	bArm2VertStn4Down_00 AT %MX26516.0 : BOOL;
	bArm2VertStn4Down_01 AT %MX26516.1 : BOOL;
	bArm2VertStn4Down_02 AT %MX26516.2 : BOOL;
	bArm2VertStn4Down_03 AT %MX26516.3 : BOOL;
	bArm2VertStn4Down_04 AT %MX26516.4 : BOOL;
	bArm2VertStn4Down_05 AT %MX26516.5 : BOOL;
	bArm2VertStn4Down_06 AT %MX26516.6 : BOOL;
	bArm2VertStn4Down_07 AT %MX26516.7 : BOOL;
	bArm2VertStn4Down_08 AT %MX26516.8 : BOOL;
	bArm2VertStn4Down_09 AT %MX26516.9 : BOOL;
	bArm2VertStn4Down_10 AT %MX26516.10 : BOOL;
	bArm2VertStn4Down_11 AT %MX26516.11 : BOOL;
	bArm2VertStn4Down_12 AT %MX26516.12 : BOOL;
	bArm2VertStn4Down_13 AT %MX26516.13 : BOOL;
	bArm2VertStn4Down_14 AT %MX26516.14 : BOOL;
	bArm2VertStn4Down_15 AT %MX26516.15 : BOOL;
	bArm2VertStn4Down_16 AT %MX26516.16 : BOOL;
	bArm2VertStn4Down_17 AT %MX26516.17 : BOOL;
	bArm2VertStn4Down_18 AT %MX26516.18 : BOOL;
	bArm2VertStn4Down_19 AT %MX26516.19 : BOOL;
	bArm2VertStn4Down_20 AT %MX26516.20 : BOOL;
	bArm2VertStn4Down_21 AT %MX26516.21 : BOOL;
	bArm2VertStn4Down_22 AT %MX26516.22 : BOOL;
	bArm2VertStn4Down_23 AT %MX26516.23 : BOOL;
	bArm2VertStn4Down_24 AT %MX26516.24 : BOOL;
	bArm2VertStn4Down_25 AT %MX26516.25 : BOOL;
	bArm2VertStn4Down_26 AT %MX26516.26 : BOOL;
	bArm2VertStn4Down_27 AT %MX26516.27 : BOOL;
	bArm2VertStn4Down_28 AT %MX26516.28 : BOOL;
	bArm2VertStn4Down_29 AT %MX26516.29 : BOOL;
	bArm2VertStn4Down_30 AT %MX26516.30 : BOOL;
	bArm2VertStn4Down_31 AT %MX26516.31 : BOOL;

	bArm2VertStn5Down_00 AT %MX26520.0 : BOOL;
	bArm2VertStn5Down_01 AT %MX26520.1 : BOOL;
	bArm2VertStn5Down_02 AT %MX26520.2 : BOOL;
	bArm2VertStn5Down_03 AT %MX26520.3 : BOOL;
	bArm2VertStn5Down_04 AT %MX26520.4 : BOOL;
	bArm2VertStn5Down_05 AT %MX26520.5 : BOOL;
	bArm2VertStn5Down_06 AT %MX26520.6 : BOOL;
	bArm2VertStn5Down_07 AT %MX26520.7 : BOOL;
	bArm2VertStn5Down_08 AT %MX26520.8 : BOOL;
	bArm2VertStn5Down_09 AT %MX26520.9 : BOOL;
	bArm2VertStn5Down_10 AT %MX26520.10 : BOOL;
	bArm2VertStn5Down_11 AT %MX26520.11 : BOOL;
	bArm2VertStn5Down_12 AT %MX26520.12 : BOOL;
	bArm2VertStn5Down_13 AT %MX26520.13 : BOOL;
	bArm2VertStn5Down_14 AT %MX26520.14 : BOOL;
	bArm2VertStn5Down_15 AT %MX26520.15 : BOOL;
	bArm2VertStn5Down_16 AT %MX26520.16 : BOOL;
	bArm2VertStn5Down_17 AT %MX26520.17 : BOOL;
	bArm2VertStn5Down_18 AT %MX26520.18 : BOOL;
	bArm2VertStn5Down_19 AT %MX26520.19 : BOOL;
	bArm2VertStn5Down_20 AT %MX26520.20 : BOOL;
	bArm2VertStn5Down_21 AT %MX26520.21 : BOOL;
	bArm2VertStn5Down_22 AT %MX26520.22 : BOOL;
	bArm2VertStn5Down_23 AT %MX26520.23 : BOOL;
	bArm2VertStn5Down_24 AT %MX26520.24 : BOOL;
	bArm2VertStn5Down_25 AT %MX26520.25 : BOOL;
	bArm2VertStn5Down_26 AT %MX26520.26 : BOOL;
	bArm2VertStn5Down_27 AT %MX26520.27 : BOOL;
	bArm2VertStn5Down_28 AT %MX26520.28 : BOOL;
	bArm2VertStn5Down_29 AT %MX26520.29 : BOOL;
	bArm2VertStn5Down_30 AT %MX26520.30 : BOOL;
	bArm2VertStn5Down_31 AT %MX26520.31 : BOOL;

	bArm2VertStn6Down_00 AT %MX26524.0 : BOOL;
	bArm2VertStn6Down_01 AT %MX26524.1 : BOOL;
	bArm2VertStn6Down_02 AT %MX26524.2 : BOOL;
	bArm2VertStn6Down_03 AT %MX26524.3 : BOOL;
	bArm2VertStn6Down_04 AT %MX26524.4 : BOOL;
	bArm2VertStn6Down_05 AT %MX26524.5 : BOOL;
	bArm2VertStn6Down_06 AT %MX26524.6 : BOOL;
	bArm2VertStn6Down_07 AT %MX26524.7 : BOOL;
	bArm2VertStn6Down_08 AT %MX26524.8 : BOOL;
	bArm2VertStn6Down_09 AT %MX26524.9 : BOOL;
	bArm2VertStn6Down_10 AT %MX26524.10 : BOOL;
	bArm2VertStn6Down_11 AT %MX26524.11 : BOOL;
	bArm2VertStn6Down_12 AT %MX26524.12 : BOOL;
	bArm2VertStn6Down_13 AT %MX26524.13 : BOOL;
	bArm2VertStn6Down_14 AT %MX26524.14 : BOOL;
	bArm2VertStn6Down_15 AT %MX26524.15 : BOOL;
	bArm2VertStn6Down_16 AT %MX26524.16 : BOOL;
	bArm2VertStn6Down_17 AT %MX26524.17 : BOOL;
	bArm2VertStn6Down_18 AT %MX26524.18 : BOOL;
	bArm2VertStn6Down_19 AT %MX26524.19 : BOOL;
	bArm2VertStn6Down_20 AT %MX26524.20 : BOOL;
	bArm2VertStn6Down_21 AT %MX26524.21 : BOOL;
	bArm2VertStn6Down_22 AT %MX26524.22 : BOOL;
	bArm2VertStn6Down_23 AT %MX26524.23 : BOOL;
	bArm2VertStn6Down_24 AT %MX26524.24 : BOOL;
	bArm2VertStn6Down_25 AT %MX26524.25 : BOOL;
	bArm2VertStn6Down_26 AT %MX26524.26 : BOOL;
	bArm2VertStn6Down_27 AT %MX26524.27 : BOOL;
	bArm2VertStn6Down_28 AT %MX26524.28 : BOOL;
	bArm2VertStn6Down_29 AT %MX26524.29 : BOOL;
	bArm2VertStn6Down_30 AT %MX26524.30 : BOOL;
	bArm2VertStn6Down_31 AT %MX26524.31 : BOOL;

	bArm2VertStn7Down_00 AT %MX26528.0 : BOOL;
	bArm2VertStn7Down_01 AT %MX26528.1 : BOOL;
	bArm2VertStn7Down_02 AT %MX26528.2 : BOOL;
	bArm2VertStn7Down_03 AT %MX26528.3 : BOOL;
	bArm2VertStn7Down_04 AT %MX26528.4 : BOOL;
	bArm2VertStn7Down_05 AT %MX26528.5 : BOOL;
	bArm2VertStn7Down_06 AT %MX26528.6 : BOOL;
	bArm2VertStn7Down_07 AT %MX26528.7 : BOOL;
	bArm2VertStn7Down_08 AT %MX26528.8 : BOOL;
	bArm2VertStn7Down_09 AT %MX26528.9 : BOOL;
	bArm2VertStn7Down_10 AT %MX26528.10 : BOOL;
	bArm2VertStn7Down_11 AT %MX26528.11 : BOOL;
	bArm2VertStn7Down_12 AT %MX26528.12 : BOOL;
	bArm2VertStn7Down_13 AT %MX26528.13 : BOOL;
	bArm2VertStn7Down_14 AT %MX26528.14 : BOOL;
	bArm2VertStn7Down_15 AT %MX26528.15 : BOOL;
	bArm2VertStn7Down_16 AT %MX26528.16 : BOOL;
	bArm2VertStn7Down_17 AT %MX26528.17 : BOOL;
	bArm2VertStn7Down_18 AT %MX26528.18 : BOOL;
	bArm2VertStn7Down_19 AT %MX26528.19 : BOOL;
	bArm2VertStn7Down_20 AT %MX26528.20 : BOOL;
	bArm2VertStn7Down_21 AT %MX26528.21 : BOOL;
	bArm2VertStn7Down_22 AT %MX26528.22 : BOOL;
	bArm2VertStn7Down_23 AT %MX26528.23 : BOOL;
	bArm2VertStn7Down_24 AT %MX26528.24 : BOOL;
	bArm2VertStn7Down_25 AT %MX26528.25 : BOOL;
	bArm2VertStn7Down_26 AT %MX26528.26 : BOOL;
	bArm2VertStn7Down_27 AT %MX26528.27 : BOOL;
	bArm2VertStn7Down_28 AT %MX26528.28 : BOOL;
	bArm2VertStn7Down_29 AT %MX26528.29 : BOOL;
	bArm2VertStn7Down_30 AT %MX26528.30 : BOOL;
	bArm2VertStn7Down_31 AT %MX26528.31 : BOOL;

	bArm2VertStn8Down_00 AT %MX26532.0 : BOOL;
	bArm2VertStn8Down_01 AT %MX26532.1 : BOOL;
	bArm2VertStn8Down_02 AT %MX26532.2 : BOOL;
	bArm2VertStn8Down_03 AT %MX26532.3 : BOOL;
	bArm2VertStn8Down_04 AT %MX26532.4 : BOOL;
	bArm2VertStn8Down_05 AT %MX26532.5 : BOOL;
	bArm2VertStn8Down_06 AT %MX26532.6 : BOOL;
	bArm2VertStn8Down_07 AT %MX26532.7 : BOOL;
	bArm2VertStn8Down_08 AT %MX26532.8 : BOOL;
	bArm2VertStn8Down_09 AT %MX26532.9 : BOOL;
	bArm2VertStn8Down_10 AT %MX26532.10 : BOOL;
	bArm2VertStn8Down_11 AT %MX26532.11 : BOOL;
	bArm2VertStn8Down_12 AT %MX26532.12 : BOOL;
	bArm2VertStn8Down_13 AT %MX26532.13 : BOOL;
	bArm2VertStn8Down_14 AT %MX26532.14 : BOOL;
	bArm2VertStn8Down_15 AT %MX26532.15 : BOOL;
	bArm2VertStn8Down_16 AT %MX26532.16 : BOOL;
	bArm2VertStn8Down_17 AT %MX26532.17 : BOOL;
	bArm2VertStn8Down_18 AT %MX26532.18 : BOOL;
	bArm2VertStn8Down_19 AT %MX26532.19 : BOOL;
	bArm2VertStn8Down_20 AT %MX26532.20 : BOOL;
	bArm2VertStn8Down_21 AT %MX26532.21 : BOOL;
	bArm2VertStn8Down_22 AT %MX26532.22 : BOOL;
	bArm2VertStn8Down_23 AT %MX26532.23 : BOOL;
	bArm2VertStn8Down_24 AT %MX26532.24 : BOOL;
	bArm2VertStn8Down_25 AT %MX26532.25 : BOOL;
	bArm2VertStn8Down_26 AT %MX26532.26 : BOOL;
	bArm2VertStn8Down_27 AT %MX26532.27 : BOOL;
	bArm2VertStn8Down_28 AT %MX26532.28 : BOOL;
	bArm2VertStn8Down_29 AT %MX26532.29 : BOOL;
	bArm2VertStn8Down_30 AT %MX26532.30 : BOOL;
	bArm2VertStn8Down_31 AT %MX26532.31 : BOOL;

	bArm2VertStn9Down_00 AT %MX26536.0 : BOOL;
	bArm2VertStn9Down_01 AT %MX26536.1 : BOOL;
	bArm2VertStn9Down_02 AT %MX26536.2 : BOOL;
	bArm2VertStn9Down_03 AT %MX26536.3 : BOOL;
	bArm2VertStn9Down_04 AT %MX26536.4 : BOOL;
	bArm2VertStn9Down_05 AT %MX26536.5 : BOOL;
	bArm2VertStn9Down_06 AT %MX26536.6 : BOOL;
	bArm2VertStn9Down_07 AT %MX26536.7 : BOOL;
	bArm2VertStn9Down_08 AT %MX26536.8 : BOOL;
	bArm2VertStn9Down_09 AT %MX26536.9 : BOOL;
	bArm2VertStn9Down_10 AT %MX26536.10 : BOOL;
	bArm2VertStn9Down_11 AT %MX26536.11 : BOOL;
	bArm2VertStn9Down_12 AT %MX26536.12 : BOOL;
	bArm2VertStn9Down_13 AT %MX26536.13 : BOOL;
	bArm2VertStn9Down_14 AT %MX26536.14 : BOOL;
	bArm2VertStn9Down_15 AT %MX26536.15 : BOOL;
	bArm2VertStn9Down_16 AT %MX26536.16 : BOOL;
	bArm2VertStn9Down_17 AT %MX26536.17 : BOOL;
	bArm2VertStn9Down_18 AT %MX26536.18 : BOOL;
	bArm2VertStn9Down_19 AT %MX26536.19 : BOOL;
	bArm2VertStn9Down_20 AT %MX26536.20 : BOOL;
	bArm2VertStn9Down_21 AT %MX26536.21 : BOOL;
	bArm2VertStn9Down_22 AT %MX26536.22 : BOOL;
	bArm2VertStn9Down_23 AT %MX26536.23 : BOOL;
	bArm2VertStn9Down_24 AT %MX26536.24 : BOOL;
	bArm2VertStn9Down_25 AT %MX26536.25 : BOOL;
	bArm2VertStn9Down_26 AT %MX26536.26 : BOOL;
	bArm2VertStn9Down_27 AT %MX26536.27 : BOOL;
	bArm2VertStn9Down_28 AT %MX26536.28 : BOOL;
	bArm2VertStn9Down_29 AT %MX26536.29 : BOOL;
	bArm2VertStn9Down_30 AT %MX26536.30 : BOOL;
	bArm2VertStn9Down_31 AT %MX26536.31 : BOOL;

	bArm2VertStn10Down_00 AT %MX26540.0 : BOOL;
	bArm2VertStn10Down_01 AT %MX26540.1 : BOOL;
	bArm2VertStn10Down_02 AT %MX26540.2 : BOOL;
	bArm2VertStn10Down_03 AT %MX26540.3 : BOOL;
	bArm2VertStn10Down_04 AT %MX26540.4 : BOOL;
	bArm2VertStn10Down_05 AT %MX26540.5 : BOOL;
	bArm2VertStn10Down_06 AT %MX26540.6 : BOOL;
	bArm2VertStn10Down_07 AT %MX26540.7 : BOOL;
	bArm2VertStn10Down_08 AT %MX26540.8 : BOOL;
	bArm2VertStn10Down_09 AT %MX26540.9 : BOOL;
	bArm2VertStn10Down_10 AT %MX26540.10 : BOOL;
	bArm2VertStn10Down_11 AT %MX26540.11 : BOOL;
	bArm2VertStn10Down_12 AT %MX26540.12 : BOOL;
	bArm2VertStn10Down_13 AT %MX26540.13 : BOOL;
	bArm2VertStn10Down_14 AT %MX26540.14 : BOOL;
	bArm2VertStn10Down_15 AT %MX26540.15 : BOOL;
	bArm2VertStn10Down_16 AT %MX26540.16 : BOOL;
	bArm2VertStn10Down_17 AT %MX26540.17 : BOOL;
	bArm2VertStn10Down_18 AT %MX26540.18 : BOOL;
	bArm2VertStn10Down_19 AT %MX26540.19 : BOOL;
	bArm2VertStn10Down_20 AT %MX26540.20 : BOOL;
	bArm2VertStn10Down_21 AT %MX26540.21 : BOOL;
	bArm2VertStn10Down_22 AT %MX26540.22 : BOOL;
	bArm2VertStn10Down_23 AT %MX26540.23 : BOOL;
	bArm2VertStn10Down_24 AT %MX26540.24 : BOOL;
	bArm2VertStn10Down_25 AT %MX26540.25 : BOOL;
	bArm2VertStn10Down_26 AT %MX26540.26 : BOOL;
	bArm2VertStn10Down_27 AT %MX26540.27 : BOOL;
	bArm2VertStn10Down_28 AT %MX26540.28 : BOOL;
	bArm2VertStn10Down_29 AT %MX26540.29 : BOOL;
	bArm2VertStn10Down_30 AT %MX26540.30 : BOOL;
	bArm2VertStn10Down_31 AT %MX26540.31 : BOOL;

	bArm2VertStn11Down_00 AT %MX26544.0 : BOOL;
	bArm2VertStn11Down_01 AT %MX26544.1 : BOOL;
	bArm2VertStn11Down_02 AT %MX26544.2 : BOOL;
	bArm2VertStn11Down_03 AT %MX26544.3 : BOOL;
	bArm2VertStn11Down_04 AT %MX26544.4 : BOOL;
	bArm2VertStn11Down_05 AT %MX26544.5 : BOOL;
	bArm2VertStn11Down_06 AT %MX26544.6 : BOOL;
	bArm2VertStn11Down_07 AT %MX26544.7 : BOOL;
	bArm2VertStn11Down_08 AT %MX26544.8 : BOOL;
	bArm2VertStn11Down_09 AT %MX26544.9 : BOOL;
	bArm2VertStn11Down_10 AT %MX26544.10 : BOOL;
	bArm2VertStn11Down_11 AT %MX26544.11 : BOOL;
	bArm2VertStn11Down_12 AT %MX26544.12 : BOOL;
	bArm2VertStn11Down_13 AT %MX26544.13 : BOOL;
	bArm2VertStn11Down_14 AT %MX26544.14 : BOOL;
	bArm2VertStn11Down_15 AT %MX26544.15 : BOOL;
	bArm2VertStn11Down_16 AT %MX26544.16 : BOOL;
	bArm2VertStn11Down_17 AT %MX26544.17 : BOOL;
	bArm2VertStn11Down_18 AT %MX26544.18 : BOOL;
	bArm2VertStn11Down_19 AT %MX26544.19 : BOOL;
	bArm2VertStn11Down_20 AT %MX26544.20 : BOOL;
	bArm2VertStn11Down_21 AT %MX26544.21 : BOOL;
	bArm2VertStn11Down_22 AT %MX26544.22 : BOOL;
	bArm2VertStn11Down_23 AT %MX26544.23 : BOOL;
	bArm2VertStn11Down_24 AT %MX26544.24 : BOOL;
	bArm2VertStn11Down_25 AT %MX26544.25 : BOOL;
	bArm2VertStn11Down_26 AT %MX26544.26 : BOOL;
	bArm2VertStn11Down_27 AT %MX26544.27 : BOOL;
	bArm2VertStn11Down_28 AT %MX26544.28 : BOOL;
	bArm2VertStn11Down_29 AT %MX26544.29 : BOOL;
	bArm2VertStn11Down_30 AT %MX26544.30 : BOOL;
	bArm2VertStn11Down_31 AT %MX26544.31 : BOOL;

	bArm2VertStn12Down_00 AT %MX26548.0 : BOOL;
	bArm2VertStn12Down_01 AT %MX26548.1 : BOOL;
	bArm2VertStn12Down_02 AT %MX26548.2 : BOOL;
	bArm2VertStn12Down_03 AT %MX26548.3 : BOOL;
	bArm2VertStn12Down_04 AT %MX26548.4 : BOOL;
	bArm2VertStn12Down_05 AT %MX26548.5 : BOOL;
	bArm2VertStn12Down_06 AT %MX26548.6 : BOOL;
	bArm2VertStn12Down_07 AT %MX26548.7 : BOOL;
	bArm2VertStn12Down_08 AT %MX26548.8 : BOOL;
	bArm2VertStn12Down_09 AT %MX26548.9 : BOOL;
	bArm2VertStn12Down_10 AT %MX26548.10 : BOOL;
	bArm2VertStn12Down_11 AT %MX26548.11 : BOOL;
	bArm2VertStn12Down_12 AT %MX26548.12 : BOOL;
	bArm2VertStn12Down_13 AT %MX26548.13 : BOOL;
	bArm2VertStn12Down_14 AT %MX26548.14 : BOOL;
	bArm2VertStn12Down_15 AT %MX26548.15 : BOOL;
	bArm2VertStn12Down_16 AT %MX26548.16 : BOOL;
	bArm2VertStn12Down_17 AT %MX26548.17 : BOOL;
	bArm2VertStn12Down_18 AT %MX26548.18 : BOOL;
	bArm2VertStn12Down_19 AT %MX26548.19 : BOOL;
	bArm2VertStn12Down_20 AT %MX26548.20 : BOOL;
	bArm2VertStn12Down_21 AT %MX26548.21 : BOOL;
	bArm2VertStn12Down_22 AT %MX26548.22 : BOOL;
	bArm2VertStn12Down_23 AT %MX26548.23 : BOOL;
	bArm2VertStn12Down_24 AT %MX26548.24 : BOOL;
	bArm2VertStn12Down_25 AT %MX26548.25 : BOOL;
	bArm2VertStn12Down_26 AT %MX26548.26 : BOOL;
	bArm2VertStn12Down_27 AT %MX26548.27 : BOOL;
	bArm2VertStn12Down_28 AT %MX26548.28 : BOOL;
	bArm2VertStn12Down_29 AT %MX26548.29 : BOOL;
	bArm2VertStn12Down_30 AT %MX26548.30 : BOOL;
	bArm2VertStn12Down_31 AT %MX26548.31 : BOOL;


(* xxxxxxxxxxxxxxxxxxxxxxxxxxxxxxxxxxxxxxx Lifter xxxxxxxxxxxxxxxxxxxxxxxxxxxxxxxxxxxxxxx*)
(*========= Up/Down LifterUp BOOL LINK with %MX31000-  =========*)

	bSlowPull2LifterStn1Up_00 AT %MX31004.0 : BOOL;
	bSlowPull2LifterStn1Up_01 AT %MX31004.1 : BOOL;
	bSlowPull2LifterStn1Up_02 AT %MX31004.2 : BOOL;
	bSlowPull2LifterStn1Up_03 AT %MX31004.3 : BOOL;
	bSlowPull2LifterStn1Up_04 AT %MX31004.4 : BOOL;
	bSlowPull2LifterStn1Up_05 AT %MX31004.5 : BOOL;
	bSlowPull2LifterStn1Up_06 AT %MX31004.6 : BOOL;
	bSlowPull2LifterStn1Up_07 AT %MX31004.7 : BOOL;
	bSlowPull2LifterStn1Up_08 AT %MX31004.8 : BOOL;
	bSlowPull2LifterStn1Up_09 AT %MX31004.9 : BOOL;
	bSlowPull2LifterStn1Up_10 AT %MX31004.10 : BOOL;
	bSlowPull2LifterStn1Up_11 AT %MX31004.11 : BOOL;
	bSlowPull2LifterStn1Up_12 AT %MX31004.12 : BOOL;
	bSlowPull2LifterStn1Up_13 AT %MX31004.13 : BOOL;
	bSlowPull2LifterStn1Up_14 AT %MX31004.14 : BOOL;
	bSlowPull2LifterStn1Up_15 AT %MX31004.15 : BOOL;
	bSlowPull2LifterStn1Up_16 AT %MX31004.16 : BOOL;
	bSlowPull2LifterStn1Up_17 AT %MX31004.17 : BOOL;
	bSlowPull2LifterStn1Up_18 AT %MX31004.18 : BOOL;
	bSlowPull2LifterStn1Up_19 AT %MX31004.19 : BOOL;
	bSlowPull2LifterStn1Up_20 AT %MX31004.20 : BOOL;
	bSlowPull2LifterStn1Up_21 AT %MX31004.21 : BOOL;
	bSlowPull2LifterStn1Up_22 AT %MX31004.22 : BOOL;
	bSlowPull2LifterStn1Up_23 AT %MX31004.23 : BOOL;
	bSlowPull2LifterStn1Up_24 AT %MX31004.24 : BOOL;
	bSlowPull2LifterStn1Up_25 AT %MX31004.25 : BOOL;
	bSlowPull2LifterStn1Up_26 AT %MX31004.26 : BOOL;
	bSlowPull2LifterStn1Up_27 AT %MX31004.27 : BOOL;
	bSlowPull2LifterStn1Up_28 AT %MX31004.28 : BOOL;
	bSlowPull2LifterStn1Up_29 AT %MX31004.29 : BOOL;
	bSlowPull2LifterStn1Up_30 AT %MX31004.30 : BOOL;
	bSlowPull2LifterStn1Up_31 AT %MX31004.31 : BOOL;

	bSlowPull2LifterStn2Up_00 AT %MX31008.0 : BOOL;
	bSlowPull2LifterStn2Up_01 AT %MX31008.1 : BOOL;
	bSlowPull2LifterStn2Up_02 AT %MX31008.2 : BOOL;
	bSlowPull2LifterStn2Up_03 AT %MX31008.3 : BOOL;
	bSlowPull2LifterStn2Up_04 AT %MX31008.4 : BOOL;
	bSlowPull2LifterStn2Up_05 AT %MX31008.5 : BOOL;
	bSlowPull2LifterStn2Up_06 AT %MX31008.6 : BOOL;
	bSlowPull2LifterStn2Up_07 AT %MX31008.7 : BOOL;
	bSlowPull2LifterStn2Up_08 AT %MX31008.8 : BOOL;
	bSlowPull2LifterStn2Up_09 AT %MX31008.9 : BOOL;
	bSlowPull2LifterStn2Up_10 AT %MX31008.10 : BOOL;
	bSlowPull2LifterStn2Up_11 AT %MX31008.11 : BOOL;
	bSlowPull2LifterStn2Up_12 AT %MX31008.12 : BOOL;
	bSlowPull2LifterStn2Up_13 AT %MX31008.13 : BOOL;
	bSlowPull2LifterStn2Up_14 AT %MX31008.14 : BOOL;
	bSlowPull2LifterStn2Up_15 AT %MX31008.15 : BOOL;
	bSlowPull2LifterStn2Up_16 AT %MX31008.16 : BOOL;
	bSlowPull2LifterStn2Up_17 AT %MX31008.17 : BOOL;
	bSlowPull2LifterStn2Up_18 AT %MX31008.18 : BOOL;
	bSlowPull2LifterStn2Up_19 AT %MX31008.19 : BOOL;
	bSlowPull2LifterStn2Up_20 AT %MX31008.20 : BOOL;
	bSlowPull2LifterStn2Up_21 AT %MX31008.21 : BOOL;
	bSlowPull2LifterStn2Up_22 AT %MX31008.22 : BOOL;
	bSlowPull2LifterStn2Up_23 AT %MX31008.23 : BOOL;
	bSlowPull2LifterStn2Up_24 AT %MX31008.24 : BOOL;
	bSlowPull2LifterStn2Up_25 AT %MX31008.25 : BOOL;
	bSlowPull2LifterStn2Up_26 AT %MX31008.26 : BOOL;
	bSlowPull2LifterStn2Up_27 AT %MX31008.27 : BOOL;
	bSlowPull2LifterStn2Up_28 AT %MX31008.28 : BOOL;
	bSlowPull2LifterStn2Up_29 AT %MX31008.29 : BOOL;
	bSlowPull2LifterStn2Up_30 AT %MX31008.30 : BOOL;
	bSlowPull2LifterStn2Up_31 AT %MX31008.31 : BOOL;

	bSlowPull2LifterStn3Up_00 AT %MX31012.0 : BOOL;
	bSlowPull2LifterStn3Up_01 AT %MX31012.1 : BOOL;
	bSlowPull2LifterStn3Up_02 AT %MX31012.2 : BOOL;
	bSlowPull2LifterStn3Up_03 AT %MX31012.3 : BOOL;
	bSlowPull2LifterStn3Up_04 AT %MX31012.4 : BOOL;
	bSlowPull2LifterStn3Up_05 AT %MX31012.5 : BOOL;
	bSlowPull2LifterStn3Up_06 AT %MX31012.6 : BOOL;
	bSlowPull2LifterStn3Up_07 AT %MX31012.7 : BOOL;
	bSlowPull2LifterStn3Up_08 AT %MX31012.8 : BOOL;
	bSlowPull2LifterStn3Up_09 AT %MX31012.9 : BOOL;
	bSlowPull2LifterStn3Up_10 AT %MX31012.10 : BOOL;
	bSlowPull2LifterStn3Up_11 AT %MX31012.11 : BOOL;
	bSlowPull2LifterStn3Up_12 AT %MX31012.12 : BOOL;
	bSlowPull2LifterStn3Up_13 AT %MX31012.13 : BOOL;
	bSlowPull2LifterStn3Up_14 AT %MX31012.14 : BOOL;
	bSlowPull2LifterStn3Up_15 AT %MX31012.15 : BOOL;
	bSlowPull2LifterStn3Up_16 AT %MX31012.16 : BOOL;
	bSlowPull2LifterStn3Up_17 AT %MX31012.17 : BOOL;
	bSlowPull2LifterStn3Up_18 AT %MX31012.18 : BOOL;
	bSlowPull2LifterStn3Up_19 AT %MX31012.19 : BOOL;
	bSlowPull2LifterStn3Up_20 AT %MX31012.20 : BOOL;
	bSlowPull2LifterStn3Up_21 AT %MX31012.21 : BOOL;
	bSlowPull2LifterStn3Up_22 AT %MX31012.22 : BOOL;
	bSlowPull2LifterStn3Up_23 AT %MX31012.23 : BOOL;
	bSlowPull2LifterStn3Up_24 AT %MX31012.24 : BOOL;
	bSlowPull2LifterStn3Up_25 AT %MX31012.25 : BOOL;
	bSlowPull2LifterStn3Up_26 AT %MX31012.26 : BOOL;
	bSlowPull2LifterStn3Up_27 AT %MX31012.27 : BOOL;
	bSlowPull2LifterStn3Up_28 AT %MX31012.28 : BOOL;
	bSlowPull2LifterStn3Up_29 AT %MX31012.29 : BOOL;
	bSlowPull2LifterStn3Up_30 AT %MX31012.30 : BOOL;
	bSlowPull2LifterStn3Up_31 AT %MX31012.31 : BOOL;

	bSlowPull2LifterStn4Up_00 AT %MX31016.0 : BOOL;
	bSlowPull2LifterStn4Up_01 AT %MX31016.1 : BOOL;
	bSlowPull2LifterStn4Up_02 AT %MX31016.2 : BOOL;
	bSlowPull2LifterStn4Up_03 AT %MX31016.3 : BOOL;
	bSlowPull2LifterStn4Up_04 AT %MX31016.4 : BOOL;
	bSlowPull2LifterStn4Up_05 AT %MX31016.5 : BOOL;
	bSlowPull2LifterStn4Up_06 AT %MX31016.6 : BOOL;
	bSlowPull2LifterStn4Up_07 AT %MX31016.7 : BOOL;
	bSlowPull2LifterStn4Up_08 AT %MX31016.8 : BOOL;
	bSlowPull2LifterStn4Up_09 AT %MX31016.9 : BOOL;
	bSlowPull2LifterStn4Up_10 AT %MX31016.10 : BOOL;
	bSlowPull2LifterStn4Up_11 AT %MX31016.11 : BOOL;
	bSlowPull2LifterStn4Up_12 AT %MX31016.12 : BOOL;
	bSlowPull2LifterStn4Up_13 AT %MX31016.13 : BOOL;
	bSlowPull2LifterStn4Up_14 AT %MX31016.14 : BOOL;
	bSlowPull2LifterStn4Up_15 AT %MX31016.15 : BOOL;
	bSlowPull2LifterStn4Up_16 AT %MX31016.16 : BOOL;
	bSlowPull2LifterStn4Up_17 AT %MX31016.17 : BOOL;
	bSlowPull2LifterStn4Up_18 AT %MX31016.18 : BOOL;
	bSlowPull2LifterStn4Up_19 AT %MX31016.19 : BOOL;
	bSlowPull2LifterStn4Up_20 AT %MX31016.20 : BOOL;
	bSlowPull2LifterStn4Up_21 AT %MX31016.21 : BOOL;
	bSlowPull2LifterStn4Up_22 AT %MX31016.22 : BOOL;
	bSlowPull2LifterStn4Up_23 AT %MX31016.23 : BOOL;
	bSlowPull2LifterStn4Up_24 AT %MX31016.24 : BOOL;
	bSlowPull2LifterStn4Up_25 AT %MX31016.25 : BOOL;
	bSlowPull2LifterStn4Up_26 AT %MX31016.26 : BOOL;
	bSlowPull2LifterStn4Up_27 AT %MX31016.27 : BOOL;
	bSlowPull2LifterStn4Up_28 AT %MX31016.28 : BOOL;
	bSlowPull2LifterStn4Up_29 AT %MX31016.29 : BOOL;
	bSlowPull2LifterStn4Up_30 AT %MX31016.30 : BOOL;
	bSlowPull2LifterStn4Up_31 AT %MX31016.31 : BOOL;

	bSlowPull2LifterStn5Up_00 AT %MX31020.0 : BOOL;
	bSlowPull2LifterStn5Up_01 AT %MX31020.1 : BOOL;
	bSlowPull2LifterStn5Up_02 AT %MX31020.2 : BOOL;
	bSlowPull2LifterStn5Up_03 AT %MX31020.3 : BOOL;
	bSlowPull2LifterStn5Up_04 AT %MX31020.4 : BOOL;
	bSlowPull2LifterStn5Up_05 AT %MX31020.5 : BOOL;
	bSlowPull2LifterStn5Up_06 AT %MX31020.6 : BOOL;
	bSlowPull2LifterStn5Up_07 AT %MX31020.7 : BOOL;
	bSlowPull2LifterStn5Up_08 AT %MX31020.8 : BOOL;
	bSlowPull2LifterStn5Up_09 AT %MX31020.9 : BOOL;
	bSlowPull2LifterStn5Up_10 AT %MX31020.10 : BOOL;
	bSlowPull2LifterStn5Up_11 AT %MX31020.11 : BOOL;
	bSlowPull2LifterStn5Up_12 AT %MX31020.12 : BOOL;
	bSlowPull2LifterStn5Up_13 AT %MX31020.13 : BOOL;
	bSlowPull2LifterStn5Up_14 AT %MX31020.14 : BOOL;
	bSlowPull2LifterStn5Up_15 AT %MX31020.15 : BOOL;
	bSlowPull2LifterStn5Up_16 AT %MX31020.16 : BOOL;
	bSlowPull2LifterStn5Up_17 AT %MX31020.17 : BOOL;
	bSlowPull2LifterStn5Up_18 AT %MX31020.18 : BOOL;
	bSlowPull2LifterStn5Up_19 AT %MX31020.19 : BOOL;
	bSlowPull2LifterStn5Up_20 AT %MX31020.20 : BOOL;
	bSlowPull2LifterStn5Up_21 AT %MX31020.21 : BOOL;
	bSlowPull2LifterStn5Up_22 AT %MX31020.22 : BOOL;
	bSlowPull2LifterStn5Up_23 AT %MX31020.23 : BOOL;
	bSlowPull2LifterStn5Up_24 AT %MX31020.24 : BOOL;
	bSlowPull2LifterStn5Up_25 AT %MX31020.25 : BOOL;
	bSlowPull2LifterStn5Up_26 AT %MX31020.26 : BOOL;
	bSlowPull2LifterStn5Up_27 AT %MX31020.27 : BOOL;
	bSlowPull2LifterStn5Up_28 AT %MX31020.28 : BOOL;
	bSlowPull2LifterStn5Up_29 AT %MX31020.29 : BOOL;
	bSlowPull2LifterStn5Up_30 AT %MX31020.30 : BOOL;
	bSlowPull2LifterStn5Up_31 AT %MX31020.31 : BOOL;

	bSlowPull2LifterStn6Up_00 AT %MX31024.0 : BOOL;
	bSlowPull2LifterStn6Up_01 AT %MX31024.1 : BOOL;
	bSlowPull2LifterStn6Up_02 AT %MX31024.2 : BOOL;
	bSlowPull2LifterStn6Up_03 AT %MX31024.3 : BOOL;
	bSlowPull2LifterStn6Up_04 AT %MX31024.4 : BOOL;
	bSlowPull2LifterStn6Up_05 AT %MX31024.5 : BOOL;
	bSlowPull2LifterStn6Up_06 AT %MX31024.6 : BOOL;
	bSlowPull2LifterStn6Up_07 AT %MX31024.7 : BOOL;
	bSlowPull2LifterStn6Up_08 AT %MX31024.8 : BOOL;
	bSlowPull2LifterStn6Up_09 AT %MX31024.9 : BOOL;
	bSlowPull2LifterStn6Up_10 AT %MX31024.10 : BOOL;
	bSlowPull2LifterStn6Up_11 AT %MX31024.11 : BOOL;
	bSlowPull2LifterStn6Up_12 AT %MX31024.12 : BOOL;
	bSlowPull2LifterStn6Up_13 AT %MX31024.13 : BOOL;
	bSlowPull2LifterStn6Up_14 AT %MX31024.14 : BOOL;
	bSlowPull2LifterStn6Up_15 AT %MX31024.15 : BOOL;
	bSlowPull2LifterStn6Up_16 AT %MX31024.16 : BOOL;
	bSlowPull2LifterStn6Up_17 AT %MX31024.17 : BOOL;
	bSlowPull2LifterStn6Up_18 AT %MX31024.18 : BOOL;
	bSlowPull2LifterStn6Up_19 AT %MX31024.19 : BOOL;
	bSlowPull2LifterStn6Up_20 AT %MX31024.20 : BOOL;
	bSlowPull2LifterStn6Up_21 AT %MX31024.21 : BOOL;
	bSlowPull2LifterStn6Up_22 AT %MX31024.22 : BOOL;
	bSlowPull2LifterStn6Up_23 AT %MX31024.23 : BOOL;
	bSlowPull2LifterStn6Up_24 AT %MX31024.24 : BOOL;
	bSlowPull2LifterStn6Up_25 AT %MX31024.25 : BOOL;
	bSlowPull2LifterStn6Up_26 AT %MX31024.26 : BOOL;
	bSlowPull2LifterStn6Up_27 AT %MX31024.27 : BOOL;
	bSlowPull2LifterStn6Up_28 AT %MX31024.28 : BOOL;
	bSlowPull2LifterStn6Up_29 AT %MX31024.29 : BOOL;
	bSlowPull2LifterStn6Up_30 AT %MX31024.30 : BOOL;
	bSlowPull2LifterStn6Up_31 AT %MX31024.31 : BOOL;

	bSlowPull2LifterStn7Up_00 AT %MX31028.0 : BOOL;
	bSlowPull2LifterStn7Up_01 AT %MX31028.1 : BOOL;
	bSlowPull2LifterStn7Up_02 AT %MX31028.2 : BOOL;
	bSlowPull2LifterStn7Up_03 AT %MX31028.3 : BOOL;
	bSlowPull2LifterStn7Up_04 AT %MX31028.4 : BOOL;
	bSlowPull2LifterStn7Up_05 AT %MX31028.5 : BOOL;
	bSlowPull2LifterStn7Up_06 AT %MX31028.6 : BOOL;
	bSlowPull2LifterStn7Up_07 AT %MX31028.7 : BOOL;
	bSlowPull2LifterStn7Up_08 AT %MX31028.8 : BOOL;
	bSlowPull2LifterStn7Up_09 AT %MX31028.9 : BOOL;
	bSlowPull2LifterStn7Up_10 AT %MX31028.10 : BOOL;
	bSlowPull2LifterStn7Up_11 AT %MX31028.11 : BOOL;
	bSlowPull2LifterStn7Up_12 AT %MX31028.12 : BOOL;
	bSlowPull2LifterStn7Up_13 AT %MX31028.13 : BOOL;
	bSlowPull2LifterStn7Up_14 AT %MX31028.14 : BOOL;
	bSlowPull2LifterStn7Up_15 AT %MX31028.15 : BOOL;
	bSlowPull2LifterStn7Up_16 AT %MX31028.16 : BOOL;
	bSlowPull2LifterStn7Up_17 AT %MX31028.17 : BOOL;
	bSlowPull2LifterStn7Up_18 AT %MX31028.18 : BOOL;
	bSlowPull2LifterStn7Up_19 AT %MX31028.19 : BOOL;
	bSlowPull2LifterStn7Up_20 AT %MX31028.20 : BOOL;
	bSlowPull2LifterStn7Up_21 AT %MX31028.21 : BOOL;
	bSlowPull2LifterStn7Up_22 AT %MX31028.22 : BOOL;
	bSlowPull2LifterStn7Up_23 AT %MX31028.23 : BOOL;
	bSlowPull2LifterStn7Up_24 AT %MX31028.24 : BOOL;
	bSlowPull2LifterStn7Up_25 AT %MX31028.25 : BOOL;
	bSlowPull2LifterStn7Up_26 AT %MX31028.26 : BOOL;
	bSlowPull2LifterStn7Up_27 AT %MX31028.27 : BOOL;
	bSlowPull2LifterStn7Up_28 AT %MX31028.28 : BOOL;
	bSlowPull2LifterStn7Up_29 AT %MX31028.29 : BOOL;
	bSlowPull2LifterStn7Up_30 AT %MX31028.30 : BOOL;
	bSlowPull2LifterStn7Up_31 AT %MX31028.31 : BOOL;

	bSlowPull2LifterStn8Up_00 AT %MX31032.0 : BOOL;
	bSlowPull2LifterStn8Up_01 AT %MX31032.1 : BOOL;
	bSlowPull2LifterStn8Up_02 AT %MX31032.2 : BOOL;
	bSlowPull2LifterStn8Up_03 AT %MX31032.3 : BOOL;
	bSlowPull2LifterStn8Up_04 AT %MX31032.4 : BOOL;
	bSlowPull2LifterStn8Up_05 AT %MX31032.5 : BOOL;
	bSlowPull2LifterStn8Up_06 AT %MX31032.6 : BOOL;
	bSlowPull2LifterStn8Up_07 AT %MX31032.7 : BOOL;
	bSlowPull2LifterStn8Up_08 AT %MX31032.8 : BOOL;
	bSlowPull2LifterStn8Up_09 AT %MX31032.9 : BOOL;
	bSlowPull2LifterStn8Up_10 AT %MX31032.10 : BOOL;
	bSlowPull2LifterStn8Up_11 AT %MX31032.11 : BOOL;
	bSlowPull2LifterStn8Up_12 AT %MX31032.12 : BOOL;
	bSlowPull2LifterStn8Up_13 AT %MX31032.13 : BOOL;
	bSlowPull2LifterStn8Up_14 AT %MX31032.14 : BOOL;
	bSlowPull2LifterStn8Up_15 AT %MX31032.15 : BOOL;
	bSlowPull2LifterStn8Up_16 AT %MX31032.16 : BOOL;
	bSlowPull2LifterStn8Up_17 AT %MX31032.17 : BOOL;
	bSlowPull2LifterStn8Up_18 AT %MX31032.18 : BOOL;
	bSlowPull2LifterStn8Up_19 AT %MX31032.19 : BOOL;
	bSlowPull2LifterStn8Up_20 AT %MX31032.20 : BOOL;
	bSlowPull2LifterStn8Up_21 AT %MX31032.21 : BOOL;
	bSlowPull2LifterStn8Up_22 AT %MX31032.22 : BOOL;
	bSlowPull2LifterStn8Up_23 AT %MX31032.23 : BOOL;
	bSlowPull2LifterStn8Up_24 AT %MX31032.24 : BOOL;
	bSlowPull2LifterStn8Up_25 AT %MX31032.25 : BOOL;
	bSlowPull2LifterStn8Up_26 AT %MX31032.26 : BOOL;
	bSlowPull2LifterStn8Up_27 AT %MX31032.27 : BOOL;
	bSlowPull2LifterStn8Up_28 AT %MX31032.28 : BOOL;
	bSlowPull2LifterStn8Up_29 AT %MX31032.29 : BOOL;
	bSlowPull2LifterStn8Up_30 AT %MX31032.30 : BOOL;
	bSlowPull2LifterStn8Up_31 AT %MX31032.31 : BOOL;

	bSlowPull2LifterStn9Up_00 AT %MX31036.0 : BOOL;
	bSlowPull2LifterStn9Up_01 AT %MX31036.1 : BOOL;
	bSlowPull2LifterStn9Up_02 AT %MX31036.2 : BOOL;
	bSlowPull2LifterStn9Up_03 AT %MX31036.3 : BOOL;
	bSlowPull2LifterStn9Up_04 AT %MX31036.4 : BOOL;
	bSlowPull2LifterStn9Up_05 AT %MX31036.5 : BOOL;
	bSlowPull2LifterStn9Up_06 AT %MX31036.6 : BOOL;
	bSlowPull2LifterStn9Up_07 AT %MX31036.7 : BOOL;
	bSlowPull2LifterStn9Up_08 AT %MX31036.8 : BOOL;
	bSlowPull2LifterStn9Up_09 AT %MX31036.9 : BOOL;
	bSlowPull2LifterStn9Up_10 AT %MX31036.10 : BOOL;
	bSlowPull2LifterStn9Up_11 AT %MX31036.11 : BOOL;
	bSlowPull2LifterStn9Up_12 AT %MX31036.12 : BOOL;
	bSlowPull2LifterStn9Up_13 AT %MX31036.13 : BOOL;
	bSlowPull2LifterStn9Up_14 AT %MX31036.14 : BOOL;
	bSlowPull2LifterStn9Up_15 AT %MX31036.15 : BOOL;
	bSlowPull2LifterStn9Up_16 AT %MX31036.16 : BOOL;
	bSlowPull2LifterStn9Up_17 AT %MX31036.17 : BOOL;
	bSlowPull2LifterStn9Up_18 AT %MX31036.18 : BOOL;
	bSlowPull2LifterStn9Up_19 AT %MX31036.19 : BOOL;
	bSlowPull2LifterStn9Up_20 AT %MX31036.20 : BOOL;
	bSlowPull2LifterStn9Up_21 AT %MX31036.21 : BOOL;
	bSlowPull2LifterStn9Up_22 AT %MX31036.22 : BOOL;
	bSlowPull2LifterStn9Up_23 AT %MX31036.23 : BOOL;
	bSlowPull2LifterStn9Up_24 AT %MX31036.24 : BOOL;
	bSlowPull2LifterStn9Up_25 AT %MX31036.25 : BOOL;
	bSlowPull2LifterStn9Up_26 AT %MX31036.26 : BOOL;
	bSlowPull2LifterStn9Up_27 AT %MX31036.27 : BOOL;
	bSlowPull2LifterStn9Up_28 AT %MX31036.28 : BOOL;
	bSlowPull2LifterStn9Up_29 AT %MX31036.29 : BOOL;
	bSlowPull2LifterStn9Up_30 AT %MX31036.30 : BOOL;
	bSlowPull2LifterStn9Up_31 AT %MX31036.31 : BOOL;

	bSlowPull2LifterStn10Up_00 AT %MX31040.0 : BOOL;
	bSlowPull2LifterStn10Up_01 AT %MX31040.1 : BOOL;
	bSlowPull2LifterStn10Up_02 AT %MX31040.2 : BOOL;
	bSlowPull2LifterStn10Up_03 AT %MX31040.3 : BOOL;
	bSlowPull2LifterStn10Up_04 AT %MX31040.4 : BOOL;
	bSlowPull2LifterStn10Up_05 AT %MX31040.5 : BOOL;
	bSlowPull2LifterStn10Up_06 AT %MX31040.6 : BOOL;
	bSlowPull2LifterStn10Up_07 AT %MX31040.7 : BOOL;
	bSlowPull2LifterStn10Up_08 AT %MX31040.8 : BOOL;
	bSlowPull2LifterStn10Up_09 AT %MX31040.9 : BOOL;
	bSlowPull2LifterStn10Up_10 AT %MX31040.10 : BOOL;
	bSlowPull2LifterStn10Up_11 AT %MX31040.11 : BOOL;
	bSlowPull2LifterStn10Up_12 AT %MX31040.12 : BOOL;
	bSlowPull2LifterStn10Up_13 AT %MX31040.13 : BOOL;
	bSlowPull2LifterStn10Up_14 AT %MX31040.14 : BOOL;
	bSlowPull2LifterStn10Up_15 AT %MX31040.15 : BOOL;
	bSlowPull2LifterStn10Up_16 AT %MX31040.16 : BOOL;
	bSlowPull2LifterStn10Up_17 AT %MX31040.17 : BOOL;
	bSlowPull2LifterStn10Up_18 AT %MX31040.18 : BOOL;
	bSlowPull2LifterStn10Up_19 AT %MX31040.19 : BOOL;
	bSlowPull2LifterStn10Up_20 AT %MX31040.20 : BOOL;
	bSlowPull2LifterStn10Up_21 AT %MX31040.21 : BOOL;
	bSlowPull2LifterStn10Up_22 AT %MX31040.22 : BOOL;
	bSlowPull2LifterStn10Up_23 AT %MX31040.23 : BOOL;
	bSlowPull2LifterStn10Up_24 AT %MX31040.24 : BOOL;
	bSlowPull2LifterStn10Up_25 AT %MX31040.25 : BOOL;
	bSlowPull2LifterStn10Up_26 AT %MX31040.26 : BOOL;
	bSlowPull2LifterStn10Up_27 AT %MX31040.27 : BOOL;
	bSlowPull2LifterStn10Up_28 AT %MX31040.28 : BOOL;
	bSlowPull2LifterStn10Up_29 AT %MX31040.29 : BOOL;
	bSlowPull2LifterStn10Up_30 AT %MX31040.30 : BOOL;
	bSlowPull2LifterStn10Up_31 AT %MX31040.31 : BOOL;

	bSlowPull2LifterStn11Up_00 AT %MX31044.0 : BOOL;
	bSlowPull2LifterStn11Up_01 AT %MX31044.1 : BOOL;
	bSlowPull2LifterStn11Up_02 AT %MX31044.2 : BOOL;
	bSlowPull2LifterStn11Up_03 AT %MX31044.3 : BOOL;
	bSlowPull2LifterStn11Up_04 AT %MX31044.4 : BOOL;
	bSlowPull2LifterStn11Up_05 AT %MX31044.5 : BOOL;
	bSlowPull2LifterStn11Up_06 AT %MX31044.6 : BOOL;
	bSlowPull2LifterStn11Up_07 AT %MX31044.7 : BOOL;
	bSlowPull2LifterStn11Up_08 AT %MX31044.8 : BOOL;
	bSlowPull2LifterStn11Up_09 AT %MX31044.9 : BOOL;
	bSlowPull2LifterStn11Up_10 AT %MX31044.10 : BOOL;
	bSlowPull2LifterStn11Up_11 AT %MX31044.11 : BOOL;
	bSlowPull2LifterStn11Up_12 AT %MX31044.12 : BOOL;
	bSlowPull2LifterStn11Up_13 AT %MX31044.13 : BOOL;
	bSlowPull2LifterStn11Up_14 AT %MX31044.14 : BOOL;
	bSlowPull2LifterStn11Up_15 AT %MX31044.15 : BOOL;
	bSlowPull2LifterStn11Up_16 AT %MX31044.16 : BOOL;
	bSlowPull2LifterStn11Up_17 AT %MX31044.17 : BOOL;
	bSlowPull2LifterStn11Up_18 AT %MX31044.18 : BOOL;
	bSlowPull2LifterStn11Up_19 AT %MX31044.19 : BOOL;
	bSlowPull2LifterStn11Up_20 AT %MX31044.20 : BOOL;
	bSlowPull2LifterStn11Up_21 AT %MX31044.21 : BOOL;
	bSlowPull2LifterStn11Up_22 AT %MX31044.22 : BOOL;
	bSlowPull2LifterStn11Up_23 AT %MX31044.23 : BOOL;
	bSlowPull2LifterStn11Up_24 AT %MX31044.24 : BOOL;
	bSlowPull2LifterStn11Up_25 AT %MX31044.25 : BOOL;
	bSlowPull2LifterStn11Up_26 AT %MX31044.26 : BOOL;
	bSlowPull2LifterStn11Up_27 AT %MX31044.27 : BOOL;
	bSlowPull2LifterStn11Up_28 AT %MX31044.28 : BOOL;
	bSlowPull2LifterStn11Up_29 AT %MX31044.29 : BOOL;
	bSlowPull2LifterStn11Up_30 AT %MX31044.30 : BOOL;
	bSlowPull2LifterStn11Up_31 AT %MX31044.31 : BOOL;

	bSlowPull2LifterStn12Up_00 AT %MX31048.0 : BOOL;
	bSlowPull2LifterStn12Up_01 AT %MX31048.1 : BOOL;
	bSlowPull2LifterStn12Up_02 AT %MX31048.2 : BOOL;
	bSlowPull2LifterStn12Up_03 AT %MX31048.3 : BOOL;
	bSlowPull2LifterStn12Up_04 AT %MX31048.4 : BOOL;
	bSlowPull2LifterStn12Up_05 AT %MX31048.5 : BOOL;
	bSlowPull2LifterStn12Up_06 AT %MX31048.6 : BOOL;
	bSlowPull2LifterStn12Up_07 AT %MX31048.7 : BOOL;
	bSlowPull2LifterStn12Up_08 AT %MX31048.8 : BOOL;
	bSlowPull2LifterStn12Up_09 AT %MX31048.9 : BOOL;
	bSlowPull2LifterStn12Up_10 AT %MX31048.10 : BOOL;
	bSlowPull2LifterStn12Up_11 AT %MX31048.11 : BOOL;
	bSlowPull2LifterStn12Up_12 AT %MX31048.12 : BOOL;
	bSlowPull2LifterStn12Up_13 AT %MX31048.13 : BOOL;
	bSlowPull2LifterStn12Up_14 AT %MX31048.14 : BOOL;
	bSlowPull2LifterStn12Up_15 AT %MX31048.15 : BOOL;
	bSlowPull2LifterStn12Up_16 AT %MX31048.16 : BOOL;
	bSlowPull2LifterStn12Up_17 AT %MX31048.17 : BOOL;
	bSlowPull2LifterStn12Up_18 AT %MX31048.18 : BOOL;
	bSlowPull2LifterStn12Up_19 AT %MX31048.19 : BOOL;
	bSlowPull2LifterStn12Up_20 AT %MX31048.20 : BOOL;
	bSlowPull2LifterStn12Up_21 AT %MX31048.21 : BOOL;
	bSlowPull2LifterStn12Up_22 AT %MX31048.22 : BOOL;
	bSlowPull2LifterStn12Up_23 AT %MX31048.23 : BOOL;
	bSlowPull2LifterStn12Up_24 AT %MX31048.24 : BOOL;
	bSlowPull2LifterStn12Up_25 AT %MX31048.25 : BOOL;
	bSlowPull2LifterStn12Up_26 AT %MX31048.26 : BOOL;
	bSlowPull2LifterStn12Up_27 AT %MX31048.27 : BOOL;
	bSlowPull2LifterStn12Up_28 AT %MX31048.28 : BOOL;
	bSlowPull2LifterStn12Up_29 AT %MX31048.29 : BOOL;
	bSlowPull2LifterStn12Up_30 AT %MX31048.30 : BOOL;
	bSlowPull2LifterStn12Up_31 AT %MX31048.31 : BOOL;


(* xxxxxxxxxxxxxxxxxxxxxxxxxxxxxxxxxxxxxxx Lifter xxxxxxxxxxxxxxxxxxxxxxxxxxxxxxxxxxxxxxx*)
(*========= Up/Down LifterDown BOOL LINK with %MX31000-  =========*)

	bSlowPull2LifterStn1Down_00 AT %MX31304.0 : BOOL;
	bSlowPull2LifterStn1Down_01 AT %MX31304.1 : BOOL;
	bSlowPull2LifterStn1Down_02 AT %MX31304.2 : BOOL;
	bSlowPull2LifterStn1Down_03 AT %MX31304.3 : BOOL;
	bSlowPull2LifterStn1Down_04 AT %MX31304.4 : BOOL;
	bSlowPull2LifterStn1Down_05 AT %MX31304.5 : BOOL;
	bSlowPull2LifterStn1Down_06 AT %MX31304.6 : BOOL;
	bSlowPull2LifterStn1Down_07 AT %MX31304.7 : BOOL;
	bSlowPull2LifterStn1Down_08 AT %MX31304.8 : BOOL;
	bSlowPull2LifterStn1Down_09 AT %MX31304.9 : BOOL;
	bSlowPull2LifterStn1Down_10 AT %MX31304.10 : BOOL;
	bSlowPull2LifterStn1Down_11 AT %MX31304.11 : BOOL;
	bSlowPull2LifterStn1Down_12 AT %MX31304.12 : BOOL;
	bSlowPull2LifterStn1Down_13 AT %MX31304.13 : BOOL;
	bSlowPull2LifterStn1Down_14 AT %MX31304.14 : BOOL;
	bSlowPull2LifterStn1Down_15 AT %MX31304.15 : BOOL;
	bSlowPull2LifterStn1Down_16 AT %MX31304.16 : BOOL;
	bSlowPull2LifterStn1Down_17 AT %MX31304.17 : BOOL;
	bSlowPull2LifterStn1Down_18 AT %MX31304.18 : BOOL;
	bSlowPull2LifterStn1Down_19 AT %MX31304.19 : BOOL;
	bSlowPull2LifterStn1Down_20 AT %MX31304.20 : BOOL;
	bSlowPull2LifterStn1Down_21 AT %MX31304.21 : BOOL;
	bSlowPull2LifterStn1Down_22 AT %MX31304.22 : BOOL;
	bSlowPull2LifterStn1Down_23 AT %MX31304.23 : BOOL;
	bSlowPull2LifterStn1Down_24 AT %MX31304.24 : BOOL;
	bSlowPull2LifterStn1Down_25 AT %MX31304.25 : BOOL;
	bSlowPull2LifterStn1Down_26 AT %MX31304.26 : BOOL;
	bSlowPull2LifterStn1Down_27 AT %MX31304.27 : BOOL;
	bSlowPull2LifterStn1Down_28 AT %MX31304.28 : BOOL;
	bSlowPull2LifterStn1Down_29 AT %MX31304.29 : BOOL;
	bSlowPull2LifterStn1Down_30 AT %MX31304.30 : BOOL;
	bSlowPull2LifterStn1Down_31 AT %MX31304.31 : BOOL;

	bSlowPull2LifterStn2Down_00 AT %MX31308.0 : BOOL;
	bSlowPull2LifterStn2Down_01 AT %MX31308.1 : BOOL;
	bSlowPull2LifterStn2Down_02 AT %MX31308.2 : BOOL;
	bSlowPull2LifterStn2Down_03 AT %MX31308.3 : BOOL;
	bSlowPull2LifterStn2Down_04 AT %MX31308.4 : BOOL;
	bSlowPull2LifterStn2Down_05 AT %MX31308.5 : BOOL;
	bSlowPull2LifterStn2Down_06 AT %MX31308.6 : BOOL;
	bSlowPull2LifterStn2Down_07 AT %MX31308.7 : BOOL;
	bSlowPull2LifterStn2Down_08 AT %MX31308.8 : BOOL;
	bSlowPull2LifterStn2Down_09 AT %MX31308.9 : BOOL;
	bSlowPull2LifterStn2Down_10 AT %MX31308.10 : BOOL;
	bSlowPull2LifterStn2Down_11 AT %MX31308.11 : BOOL;
	bSlowPull2LifterStn2Down_12 AT %MX31308.12 : BOOL;
	bSlowPull2LifterStn2Down_13 AT %MX31308.13 : BOOL;
	bSlowPull2LifterStn2Down_14 AT %MX31308.14 : BOOL;
	bSlowPull2LifterStn2Down_15 AT %MX31308.15 : BOOL;
	bSlowPull2LifterStn2Down_16 AT %MX31308.16 : BOOL;
	bSlowPull2LifterStn2Down_17 AT %MX31308.17 : BOOL;
	bSlowPull2LifterStn2Down_18 AT %MX31308.18 : BOOL;
	bSlowPull2LifterStn2Down_19 AT %MX31308.19 : BOOL;
	bSlowPull2LifterStn2Down_20 AT %MX31308.20 : BOOL;
	bSlowPull2LifterStn2Down_21 AT %MX31308.21 : BOOL;
	bSlowPull2LifterStn2Down_22 AT %MX31308.22 : BOOL;
	bSlowPull2LifterStn2Down_23 AT %MX31308.23 : BOOL;
	bSlowPull2LifterStn2Down_24 AT %MX31308.24 : BOOL;
	bSlowPull2LifterStn2Down_25 AT %MX31308.25 : BOOL;
	bSlowPull2LifterStn2Down_26 AT %MX31308.26 : BOOL;
	bSlowPull2LifterStn2Down_27 AT %MX31308.27 : BOOL;
	bSlowPull2LifterStn2Down_28 AT %MX31308.28 : BOOL;
	bSlowPull2LifterStn2Down_29 AT %MX31308.29 : BOOL;
	bSlowPull2LifterStn2Down_30 AT %MX31308.30 : BOOL;
	bSlowPull2LifterStn2Down_31 AT %MX31308.31 : BOOL;

	bSlowPull2LifterStn3Down_00 AT %MX31312.0 : BOOL;
	bSlowPull2LifterStn3Down_01 AT %MX31312.1 : BOOL;
	bSlowPull2LifterStn3Down_02 AT %MX31312.2 : BOOL;
	bSlowPull2LifterStn3Down_03 AT %MX31312.3 : BOOL;
	bSlowPull2LifterStn3Down_04 AT %MX31312.4 : BOOL;
	bSlowPull2LifterStn3Down_05 AT %MX31312.5 : BOOL;
	bSlowPull2LifterStn3Down_06 AT %MX31312.6 : BOOL;
	bSlowPull2LifterStn3Down_07 AT %MX31312.7 : BOOL;
	bSlowPull2LifterStn3Down_08 AT %MX31312.8 : BOOL;
	bSlowPull2LifterStn3Down_09 AT %MX31312.9 : BOOL;
	bSlowPull2LifterStn3Down_10 AT %MX31312.10 : BOOL;
	bSlowPull2LifterStn3Down_11 AT %MX31312.11 : BOOL;
	bSlowPull2LifterStn3Down_12 AT %MX31312.12 : BOOL;
	bSlowPull2LifterStn3Down_13 AT %MX31312.13 : BOOL;
	bSlowPull2LifterStn3Down_14 AT %MX31312.14 : BOOL;
	bSlowPull2LifterStn3Down_15 AT %MX31312.15 : BOOL;
	bSlowPull2LifterStn3Down_16 AT %MX31312.16 : BOOL;
	bSlowPull2LifterStn3Down_17 AT %MX31312.17 : BOOL;
	bSlowPull2LifterStn3Down_18 AT %MX31312.18 : BOOL;
	bSlowPull2LifterStn3Down_19 AT %MX31312.19 : BOOL;
	bSlowPull2LifterStn3Down_20 AT %MX31312.20 : BOOL;
	bSlowPull2LifterStn3Down_21 AT %MX31312.21 : BOOL;
	bSlowPull2LifterStn3Down_22 AT %MX31312.22 : BOOL;
	bSlowPull2LifterStn3Down_23 AT %MX31312.23 : BOOL;
	bSlowPull2LifterStn3Down_24 AT %MX31312.24 : BOOL;
	bSlowPull2LifterStn3Down_25 AT %MX31312.25 : BOOL;
	bSlowPull2LifterStn3Down_26 AT %MX31312.26 : BOOL;
	bSlowPull2LifterStn3Down_27 AT %MX31312.27 : BOOL;
	bSlowPull2LifterStn3Down_28 AT %MX31312.28 : BOOL;
	bSlowPull2LifterStn3Down_29 AT %MX31312.29 : BOOL;
	bSlowPull2LifterStn3Down_30 AT %MX31312.30 : BOOL;
	bSlowPull2LifterStn3Down_31 AT %MX31312.31 : BOOL;

	bSlowPull2LifterStn4Down_00 AT %MX31316.0 : BOOL;
	bSlowPull2LifterStn4Down_01 AT %MX31316.1 : BOOL;
	bSlowPull2LifterStn4Down_02 AT %MX31316.2 : BOOL;
	bSlowPull2LifterStn4Down_03 AT %MX31316.3 : BOOL;
	bSlowPull2LifterStn4Down_04 AT %MX31316.4 : BOOL;
	bSlowPull2LifterStn4Down_05 AT %MX31316.5 : BOOL;
	bSlowPull2LifterStn4Down_06 AT %MX31316.6 : BOOL;
	bSlowPull2LifterStn4Down_07 AT %MX31316.7 : BOOL;
	bSlowPull2LifterStn4Down_08 AT %MX31316.8 : BOOL;
	bSlowPull2LifterStn4Down_09 AT %MX31316.9 : BOOL;
	bSlowPull2LifterStn4Down_10 AT %MX31316.10 : BOOL;
	bSlowPull2LifterStn4Down_11 AT %MX31316.11 : BOOL;
	bSlowPull2LifterStn4Down_12 AT %MX31316.12 : BOOL;
	bSlowPull2LifterStn4Down_13 AT %MX31316.13 : BOOL;
	bSlowPull2LifterStn4Down_14 AT %MX31316.14 : BOOL;
	bSlowPull2LifterStn4Down_15 AT %MX31316.15 : BOOL;
	bSlowPull2LifterStn4Down_16 AT %MX31316.16 : BOOL;
	bSlowPull2LifterStn4Down_17 AT %MX31316.17 : BOOL;
	bSlowPull2LifterStn4Down_18 AT %MX31316.18 : BOOL;
	bSlowPull2LifterStn4Down_19 AT %MX31316.19 : BOOL;
	bSlowPull2LifterStn4Down_20 AT %MX31316.20 : BOOL;
	bSlowPull2LifterStn4Down_21 AT %MX31316.21 : BOOL;
	bSlowPull2LifterStn4Down_22 AT %MX31316.22 : BOOL;
	bSlowPull2LifterStn4Down_23 AT %MX31316.23 : BOOL;
	bSlowPull2LifterStn4Down_24 AT %MX31316.24 : BOOL;
	bSlowPull2LifterStn4Down_25 AT %MX31316.25 : BOOL;
	bSlowPull2LifterStn4Down_26 AT %MX31316.26 : BOOL;
	bSlowPull2LifterStn4Down_27 AT %MX31316.27 : BOOL;
	bSlowPull2LifterStn4Down_28 AT %MX31316.28 : BOOL;
	bSlowPull2LifterStn4Down_29 AT %MX31316.29 : BOOL;
	bSlowPull2LifterStn4Down_30 AT %MX31316.30 : BOOL;
	bSlowPull2LifterStn4Down_31 AT %MX31316.31 : BOOL;

	bSlowPull2LifterStn5Down_00 AT %MX31320.0 : BOOL;
	bSlowPull2LifterStn5Down_01 AT %MX31320.1 : BOOL;
	bSlowPull2LifterStn5Down_02 AT %MX31320.2 : BOOL;
	bSlowPull2LifterStn5Down_03 AT %MX31320.3 : BOOL;
	bSlowPull2LifterStn5Down_04 AT %MX31320.4 : BOOL;
	bSlowPull2LifterStn5Down_05 AT %MX31320.5 : BOOL;
	bSlowPull2LifterStn5Down_06 AT %MX31320.6 : BOOL;
	bSlowPull2LifterStn5Down_07 AT %MX31320.7 : BOOL;
	bSlowPull2LifterStn5Down_08 AT %MX31320.8 : BOOL;
	bSlowPull2LifterStn5Down_09 AT %MX31320.9 : BOOL;
	bSlowPull2LifterStn5Down_10 AT %MX31320.10 : BOOL;
	bSlowPull2LifterStn5Down_11 AT %MX31320.11 : BOOL;
	bSlowPull2LifterStn5Down_12 AT %MX31320.12 : BOOL;
	bSlowPull2LifterStn5Down_13 AT %MX31320.13 : BOOL;
	bSlowPull2LifterStn5Down_14 AT %MX31320.14 : BOOL;
	bSlowPull2LifterStn5Down_15 AT %MX31320.15 : BOOL;
	bSlowPull2LifterStn5Down_16 AT %MX31320.16 : BOOL;
	bSlowPull2LifterStn5Down_17 AT %MX31320.17 : BOOL;
	bSlowPull2LifterStn5Down_18 AT %MX31320.18 : BOOL;
	bSlowPull2LifterStn5Down_19 AT %MX31320.19 : BOOL;
	bSlowPull2LifterStn5Down_20 AT %MX31320.20 : BOOL;
	bSlowPull2LifterStn5Down_21 AT %MX31320.21 : BOOL;
	bSlowPull2LifterStn5Down_22 AT %MX31320.22 : BOOL;
	bSlowPull2LifterStn5Down_23 AT %MX31320.23 : BOOL;
	bSlowPull2LifterStn5Down_24 AT %MX31320.24 : BOOL;
	bSlowPull2LifterStn5Down_25 AT %MX31320.25 : BOOL;
	bSlowPull2LifterStn5Down_26 AT %MX31320.26 : BOOL;
	bSlowPull2LifterStn5Down_27 AT %MX31320.27 : BOOL;
	bSlowPull2LifterStn5Down_28 AT %MX31320.28 : BOOL;
	bSlowPull2LifterStn5Down_29 AT %MX31320.29 : BOOL;
	bSlowPull2LifterStn5Down_30 AT %MX31320.30 : BOOL;
	bSlowPull2LifterStn5Down_31 AT %MX31320.31 : BOOL;

	bSlowPull2LifterStn6Down_00 AT %MX31324.0 : BOOL;
	bSlowPull2LifterStn6Down_01 AT %MX31324.1 : BOOL;
	bSlowPull2LifterStn6Down_02 AT %MX31324.2 : BOOL;
	bSlowPull2LifterStn6Down_03 AT %MX31324.3 : BOOL;
	bSlowPull2LifterStn6Down_04 AT %MX31324.4 : BOOL;
	bSlowPull2LifterStn6Down_05 AT %MX31324.5 : BOOL;
	bSlowPull2LifterStn6Down_06 AT %MX31324.6 : BOOL;
	bSlowPull2LifterStn6Down_07 AT %MX31324.7 : BOOL;
	bSlowPull2LifterStn6Down_08 AT %MX31324.8 : BOOL;
	bSlowPull2LifterStn6Down_09 AT %MX31324.9 : BOOL;
	bSlowPull2LifterStn6Down_10 AT %MX31324.10 : BOOL;
	bSlowPull2LifterStn6Down_11 AT %MX31324.11 : BOOL;
	bSlowPull2LifterStn6Down_12 AT %MX31324.12 : BOOL;
	bSlowPull2LifterStn6Down_13 AT %MX31324.13 : BOOL;
	bSlowPull2LifterStn6Down_14 AT %MX31324.14 : BOOL;
	bSlowPull2LifterStn6Down_15 AT %MX31324.15 : BOOL;
	bSlowPull2LifterStn6Down_16 AT %MX31324.16 : BOOL;
	bSlowPull2LifterStn6Down_17 AT %MX31324.17 : BOOL;
	bSlowPull2LifterStn6Down_18 AT %MX31324.18 : BOOL;
	bSlowPull2LifterStn6Down_19 AT %MX31324.19 : BOOL;
	bSlowPull2LifterStn6Down_20 AT %MX31324.20 : BOOL;
	bSlowPull2LifterStn6Down_21 AT %MX31324.21 : BOOL;
	bSlowPull2LifterStn6Down_22 AT %MX31324.22 : BOOL;
	bSlowPull2LifterStn6Down_23 AT %MX31324.23 : BOOL;
	bSlowPull2LifterStn6Down_24 AT %MX31324.24 : BOOL;
	bSlowPull2LifterStn6Down_25 AT %MX31324.25 : BOOL;
	bSlowPull2LifterStn6Down_26 AT %MX31324.26 : BOOL;
	bSlowPull2LifterStn6Down_27 AT %MX31324.27 : BOOL;
	bSlowPull2LifterStn6Down_28 AT %MX31324.28 : BOOL;
	bSlowPull2LifterStn6Down_29 AT %MX31324.29 : BOOL;
	bSlowPull2LifterStn6Down_30 AT %MX31324.30 : BOOL;
	bSlowPull2LifterStn6Down_31 AT %MX31324.31 : BOOL;

	bSlowPull2LifterStn7Down_00 AT %MX31328.0 : BOOL;
	bSlowPull2LifterStn7Down_01 AT %MX31328.1 : BOOL;
	bSlowPull2LifterStn7Down_02 AT %MX31328.2 : BOOL;
	bSlowPull2LifterStn7Down_03 AT %MX31328.3 : BOOL;
	bSlowPull2LifterStn7Down_04 AT %MX31328.4 : BOOL;
	bSlowPull2LifterStn7Down_05 AT %MX31328.5 : BOOL;
	bSlowPull2LifterStn7Down_06 AT %MX31328.6 : BOOL;
	bSlowPull2LifterStn7Down_07 AT %MX31328.7 : BOOL;
	bSlowPull2LifterStn7Down_08 AT %MX31328.8 : BOOL;
	bSlowPull2LifterStn7Down_09 AT %MX31328.9 : BOOL;
	bSlowPull2LifterStn7Down_10 AT %MX31328.10 : BOOL;
	bSlowPull2LifterStn7Down_11 AT %MX31328.11 : BOOL;
	bSlowPull2LifterStn7Down_12 AT %MX31328.12 : BOOL;
	bSlowPull2LifterStn7Down_13 AT %MX31328.13 : BOOL;
	bSlowPull2LifterStn7Down_14 AT %MX31328.14 : BOOL;
	bSlowPull2LifterStn7Down_15 AT %MX31328.15 : BOOL;
	bSlowPull2LifterStn7Down_16 AT %MX31328.16 : BOOL;
	bSlowPull2LifterStn7Down_17 AT %MX31328.17 : BOOL;
	bSlowPull2LifterStn7Down_18 AT %MX31328.18 : BOOL;
	bSlowPull2LifterStn7Down_19 AT %MX31328.19 : BOOL;
	bSlowPull2LifterStn7Down_20 AT %MX31328.20 : BOOL;
	bSlowPull2LifterStn7Down_21 AT %MX31328.21 : BOOL;
	bSlowPull2LifterStn7Down_22 AT %MX31328.22 : BOOL;
	bSlowPull2LifterStn7Down_23 AT %MX31328.23 : BOOL;
	bSlowPull2LifterStn7Down_24 AT %MX31328.24 : BOOL;
	bSlowPull2LifterStn7Down_25 AT %MX31328.25 : BOOL;
	bSlowPull2LifterStn7Down_26 AT %MX31328.26 : BOOL;
	bSlowPull2LifterStn7Down_27 AT %MX31328.27 : BOOL;
	bSlowPull2LifterStn7Down_28 AT %MX31328.28 : BOOL;
	bSlowPull2LifterStn7Down_29 AT %MX31328.29 : BOOL;
	bSlowPull2LifterStn7Down_30 AT %MX31328.30 : BOOL;
	bSlowPull2LifterStn7Down_31 AT %MX31328.31 : BOOL;

	bSlowPull2LifterStn8Down_00 AT %MX31332.0 : BOOL;
	bSlowPull2LifterStn8Down_01 AT %MX31332.1 : BOOL;
	bSlowPull2LifterStn8Down_02 AT %MX31332.2 : BOOL;
	bSlowPull2LifterStn8Down_03 AT %MX31332.3 : BOOL;
	bSlowPull2LifterStn8Down_04 AT %MX31332.4 : BOOL;
	bSlowPull2LifterStn8Down_05 AT %MX31332.5 : BOOL;
	bSlowPull2LifterStn8Down_06 AT %MX31332.6 : BOOL;
	bSlowPull2LifterStn8Down_07 AT %MX31332.7 : BOOL;
	bSlowPull2LifterStn8Down_08 AT %MX31332.8 : BOOL;
	bSlowPull2LifterStn8Down_09 AT %MX31332.9 : BOOL;
	bSlowPull2LifterStn8Down_10 AT %MX31332.10 : BOOL;
	bSlowPull2LifterStn8Down_11 AT %MX31332.11 : BOOL;
	bSlowPull2LifterStn8Down_12 AT %MX31332.12 : BOOL;
	bSlowPull2LifterStn8Down_13 AT %MX31332.13 : BOOL;
	bSlowPull2LifterStn8Down_14 AT %MX31332.14 : BOOL;
	bSlowPull2LifterStn8Down_15 AT %MX31332.15 : BOOL;
	bSlowPull2LifterStn8Down_16 AT %MX31332.16 : BOOL;
	bSlowPull2LifterStn8Down_17 AT %MX31332.17 : BOOL;
	bSlowPull2LifterStn8Down_18 AT %MX31332.18 : BOOL;
	bSlowPull2LifterStn8Down_19 AT %MX31332.19 : BOOL;
	bSlowPull2LifterStn8Down_20 AT %MX31332.20 : BOOL;
	bSlowPull2LifterStn8Down_21 AT %MX31332.21 : BOOL;
	bSlowPull2LifterStn8Down_22 AT %MX31332.22 : BOOL;
	bSlowPull2LifterStn8Down_23 AT %MX31332.23 : BOOL;
	bSlowPull2LifterStn8Down_24 AT %MX31332.24 : BOOL;
	bSlowPull2LifterStn8Down_25 AT %MX31332.25 : BOOL;
	bSlowPull2LifterStn8Down_26 AT %MX31332.26 : BOOL;
	bSlowPull2LifterStn8Down_27 AT %MX31332.27 : BOOL;
	bSlowPull2LifterStn8Down_28 AT %MX31332.28 : BOOL;
	bSlowPull2LifterStn8Down_29 AT %MX31332.29 : BOOL;
	bSlowPull2LifterStn8Down_30 AT %MX31332.30 : BOOL;
	bSlowPull2LifterStn8Down_31 AT %MX31332.31 : BOOL;

	bSlowPull2LifterStn9Down_00 AT %MX31336.0 : BOOL;
	bSlowPull2LifterStn9Down_01 AT %MX31336.1 : BOOL;
	bSlowPull2LifterStn9Down_02 AT %MX31336.2 : BOOL;
	bSlowPull2LifterStn9Down_03 AT %MX31336.3 : BOOL;
	bSlowPull2LifterStn9Down_04 AT %MX31336.4 : BOOL;
	bSlowPull2LifterStn9Down_05 AT %MX31336.5 : BOOL;
	bSlowPull2LifterStn9Down_06 AT %MX31336.6 : BOOL;
	bSlowPull2LifterStn9Down_07 AT %MX31336.7 : BOOL;
	bSlowPull2LifterStn9Down_08 AT %MX31336.8 : BOOL;
	bSlowPull2LifterStn9Down_09 AT %MX31336.9 : BOOL;
	bSlowPull2LifterStn9Down_10 AT %MX31336.10 : BOOL;
	bSlowPull2LifterStn9Down_11 AT %MX31336.11 : BOOL;
	bSlowPull2LifterStn9Down_12 AT %MX31336.12 : BOOL;
	bSlowPull2LifterStn9Down_13 AT %MX31336.13 : BOOL;
	bSlowPull2LifterStn9Down_14 AT %MX31336.14 : BOOL;
	bSlowPull2LifterStn9Down_15 AT %MX31336.15 : BOOL;
	bSlowPull2LifterStn9Down_16 AT %MX31336.16 : BOOL;
	bSlowPull2LifterStn9Down_17 AT %MX31336.17 : BOOL;
	bSlowPull2LifterStn9Down_18 AT %MX31336.18 : BOOL;
	bSlowPull2LifterStn9Down_19 AT %MX31336.19 : BOOL;
	bSlowPull2LifterStn9Down_20 AT %MX31336.20 : BOOL;
	bSlowPull2LifterStn9Down_21 AT %MX31336.21 : BOOL;
	bSlowPull2LifterStn9Down_22 AT %MX31336.22 : BOOL;
	bSlowPull2LifterStn9Down_23 AT %MX31336.23 : BOOL;
	bSlowPull2LifterStn9Down_24 AT %MX31336.24 : BOOL;
	bSlowPull2LifterStn9Down_25 AT %MX31336.25 : BOOL;
	bSlowPull2LifterStn9Down_26 AT %MX31336.26 : BOOL;
	bSlowPull2LifterStn9Down_27 AT %MX31336.27 : BOOL;
	bSlowPull2LifterStn9Down_28 AT %MX31336.28 : BOOL;
	bSlowPull2LifterStn9Down_29 AT %MX31336.29 : BOOL;
	bSlowPull2LifterStn9Down_30 AT %MX31336.30 : BOOL;
	bSlowPull2LifterStn9Down_31 AT %MX31336.31 : BOOL;

	bSlowPull2LifterStn10Down_00 AT %MX31340.0 : BOOL;
	bSlowPull2LifterStn10Down_01 AT %MX31340.1 : BOOL;
	bSlowPull2LifterStn10Down_02 AT %MX31340.2 : BOOL;
	bSlowPull2LifterStn10Down_03 AT %MX31340.3 : BOOL;
	bSlowPull2LifterStn10Down_04 AT %MX31340.4 : BOOL;
	bSlowPull2LifterStn10Down_05 AT %MX31340.5 : BOOL;
	bSlowPull2LifterStn10Down_06 AT %MX31340.6 : BOOL;
	bSlowPull2LifterStn10Down_07 AT %MX31340.7 : BOOL;
	bSlowPull2LifterStn10Down_08 AT %MX31340.8 : BOOL;
	bSlowPull2LifterStn10Down_09 AT %MX31340.9 : BOOL;
	bSlowPull2LifterStn10Down_10 AT %MX31340.10 : BOOL;
	bSlowPull2LifterStn10Down_11 AT %MX31340.11 : BOOL;
	bSlowPull2LifterStn10Down_12 AT %MX31340.12 : BOOL;
	bSlowPull2LifterStn10Down_13 AT %MX31340.13 : BOOL;
	bSlowPull2LifterStn10Down_14 AT %MX31340.14 : BOOL;
	bSlowPull2LifterStn10Down_15 AT %MX31340.15 : BOOL;
	bSlowPull2LifterStn10Down_16 AT %MX31340.16 : BOOL;
	bSlowPull2LifterStn10Down_17 AT %MX31340.17 : BOOL;
	bSlowPull2LifterStn10Down_18 AT %MX31340.18 : BOOL;
	bSlowPull2LifterStn10Down_19 AT %MX31340.19 : BOOL;
	bSlowPull2LifterStn10Down_20 AT %MX31340.20 : BOOL;
	bSlowPull2LifterStn10Down_21 AT %MX31340.21 : BOOL;
	bSlowPull2LifterStn10Down_22 AT %MX31340.22 : BOOL;
	bSlowPull2LifterStn10Down_23 AT %MX31340.23 : BOOL;
	bSlowPull2LifterStn10Down_24 AT %MX31340.24 : BOOL;
	bSlowPull2LifterStn10Down_25 AT %MX31340.25 : BOOL;
	bSlowPull2LifterStn10Down_26 AT %MX31340.26 : BOOL;
	bSlowPull2LifterStn10Down_27 AT %MX31340.27 : BOOL;
	bSlowPull2LifterStn10Down_28 AT %MX31340.28 : BOOL;
	bSlowPull2LifterStn10Down_29 AT %MX31340.29 : BOOL;
	bSlowPull2LifterStn10Down_30 AT %MX31340.30 : BOOL;
	bSlowPull2LifterStn10Down_31 AT %MX31340.31 : BOOL;

	bSlowPull2LifterStn11Down_00 AT %MX31344.0 : BOOL;
	bSlowPull2LifterStn11Down_01 AT %MX31344.1 : BOOL;
	bSlowPull2LifterStn11Down_02 AT %MX31344.2 : BOOL;
	bSlowPull2LifterStn11Down_03 AT %MX31344.3 : BOOL;
	bSlowPull2LifterStn11Down_04 AT %MX31344.4 : BOOL;
	bSlowPull2LifterStn11Down_05 AT %MX31344.5 : BOOL;
	bSlowPull2LifterStn11Down_06 AT %MX31344.6 : BOOL;
	bSlowPull2LifterStn11Down_07 AT %MX31344.7 : BOOL;
	bSlowPull2LifterStn11Down_08 AT %MX31344.8 : BOOL;
	bSlowPull2LifterStn11Down_09 AT %MX31344.9 : BOOL;
	bSlowPull2LifterStn11Down_10 AT %MX31344.10 : BOOL;
	bSlowPull2LifterStn11Down_11 AT %MX31344.11 : BOOL;
	bSlowPull2LifterStn11Down_12 AT %MX31344.12 : BOOL;
	bSlowPull2LifterStn11Down_13 AT %MX31344.13 : BOOL;
	bSlowPull2LifterStn11Down_14 AT %MX31344.14 : BOOL;
	bSlowPull2LifterStn11Down_15 AT %MX31344.15 : BOOL;
	bSlowPull2LifterStn11Down_16 AT %MX31344.16 : BOOL;
	bSlowPull2LifterStn11Down_17 AT %MX31344.17 : BOOL;
	bSlowPull2LifterStn11Down_18 AT %MX31344.18 : BOOL;
	bSlowPull2LifterStn11Down_19 AT %MX31344.19 : BOOL;
	bSlowPull2LifterStn11Down_20 AT %MX31344.20 : BOOL;
	bSlowPull2LifterStn11Down_21 AT %MX31344.21 : BOOL;
	bSlowPull2LifterStn11Down_22 AT %MX31344.22 : BOOL;
	bSlowPull2LifterStn11Down_23 AT %MX31344.23 : BOOL;
	bSlowPull2LifterStn11Down_24 AT %MX31344.24 : BOOL;
	bSlowPull2LifterStn11Down_25 AT %MX31344.25 : BOOL;
	bSlowPull2LifterStn11Down_26 AT %MX31344.26 : BOOL;
	bSlowPull2LifterStn11Down_27 AT %MX31344.27 : BOOL;
	bSlowPull2LifterStn11Down_28 AT %MX31344.28 : BOOL;
	bSlowPull2LifterStn11Down_29 AT %MX31344.29 : BOOL;
	bSlowPull2LifterStn11Down_30 AT %MX31344.30 : BOOL;
	bSlowPull2LifterStn11Down_31 AT %MX31344.31 : BOOL;

	bSlowPull2LifterStn12Down_00 AT %MX31348.0 : BOOL;
	bSlowPull2LifterStn12Down_01 AT %MX31348.1 : BOOL;
	bSlowPull2LifterStn12Down_02 AT %MX31348.2 : BOOL;
	bSlowPull2LifterStn12Down_03 AT %MX31348.3 : BOOL;
	bSlowPull2LifterStn12Down_04 AT %MX31348.4 : BOOL;
	bSlowPull2LifterStn12Down_05 AT %MX31348.5 : BOOL;
	bSlowPull2LifterStn12Down_06 AT %MX31348.6 : BOOL;
	bSlowPull2LifterStn12Down_07 AT %MX31348.7 : BOOL;
	bSlowPull2LifterStn12Down_08 AT %MX31348.8 : BOOL;
	bSlowPull2LifterStn12Down_09 AT %MX31348.9 : BOOL;
	bSlowPull2LifterStn12Down_10 AT %MX31348.10 : BOOL;
	bSlowPull2LifterStn12Down_11 AT %MX31348.11 : BOOL;
	bSlowPull2LifterStn12Down_12 AT %MX31348.12 : BOOL;
	bSlowPull2LifterStn12Down_13 AT %MX31348.13 : BOOL;
	bSlowPull2LifterStn12Down_14 AT %MX31348.14 : BOOL;
	bSlowPull2LifterStn12Down_15 AT %MX31348.15 : BOOL;
	bSlowPull2LifterStn12Down_16 AT %MX31348.16 : BOOL;
	bSlowPull2LifterStn12Down_17 AT %MX31348.17 : BOOL;
	bSlowPull2LifterStn12Down_18 AT %MX31348.18 : BOOL;
	bSlowPull2LifterStn12Down_19 AT %MX31348.19 : BOOL;
	bSlowPull2LifterStn12Down_20 AT %MX31348.20 : BOOL;
	bSlowPull2LifterStn12Down_21 AT %MX31348.21 : BOOL;
	bSlowPull2LifterStn12Down_22 AT %MX31348.22 : BOOL;
	bSlowPull2LifterStn12Down_23 AT %MX31348.23 : BOOL;
	bSlowPull2LifterStn12Down_24 AT %MX31348.24 : BOOL;
	bSlowPull2LifterStn12Down_25 AT %MX31348.25 : BOOL;
	bSlowPull2LifterStn12Down_26 AT %MX31348.26 : BOOL;
	bSlowPull2LifterStn12Down_27 AT %MX31348.27 : BOOL;
	bSlowPull2LifterStn12Down_28 AT %MX31348.28 : BOOL;
	bSlowPull2LifterStn12Down_29 AT %MX31348.29 : BOOL;
	bSlowPull2LifterStn12Down_30 AT %MX31348.30 : BOOL;
	bSlowPull2LifterStn12Down_31 AT %MX31348.31 : BOOL;


(* xxxxxxxxxxxxxxxxxxxxxxxxxxxxxxxxxxxxxxx Lifter xxxxxxxxxxxxxxxxxxxxxxxxxxxxxxxxxxxxxxx*)
(*========= Up/Down LifterAgiUp BOOL LINK with %MX31000-  =========*)

	bSlowPull2LifterStn1AgiUp_00 AT %MX31104.0 : BOOL;
	bSlowPull2LifterStn1AgiUp_01 AT %MX31104.1 : BOOL;
	bSlowPull2LifterStn1AgiUp_02 AT %MX31104.2 : BOOL;
	bSlowPull2LifterStn1AgiUp_03 AT %MX31104.3 : BOOL;
	bSlowPull2LifterStn1AgiUp_04 AT %MX31104.4 : BOOL;
	bSlowPull2LifterStn1AgiUp_05 AT %MX31104.5 : BOOL;
	bSlowPull2LifterStn1AgiUp_06 AT %MX31104.6 : BOOL;
	bSlowPull2LifterStn1AgiUp_07 AT %MX31104.7 : BOOL;
	bSlowPull2LifterStn1AgiUp_08 AT %MX31104.8 : BOOL;
	bSlowPull2LifterStn1AgiUp_09 AT %MX31104.9 : BOOL;
	bSlowPull2LifterStn1AgiUp_10 AT %MX31104.10 : BOOL;
	bSlowPull2LifterStn1AgiUp_11 AT %MX31104.11 : BOOL;
	bSlowPull2LifterStn1AgiUp_12 AT %MX31104.12 : BOOL;
	bSlowPull2LifterStn1AgiUp_13 AT %MX31104.13 : BOOL;
	bSlowPull2LifterStn1AgiUp_14 AT %MX31104.14 : BOOL;
	bSlowPull2LifterStn1AgiUp_15 AT %MX31104.15 : BOOL;
	bSlowPull2LifterStn1AgiUp_16 AT %MX31104.16 : BOOL;
	bSlowPull2LifterStn1AgiUp_17 AT %MX31104.17 : BOOL;
	bSlowPull2LifterStn1AgiUp_18 AT %MX31104.18 : BOOL;
	bSlowPull2LifterStn1AgiUp_19 AT %MX31104.19 : BOOL;
	bSlowPull2LifterStn1AgiUp_20 AT %MX31104.20 : BOOL;
	bSlowPull2LifterStn1AgiUp_21 AT %MX31104.21 : BOOL;
	bSlowPull2LifterStn1AgiUp_22 AT %MX31104.22 : BOOL;
	bSlowPull2LifterStn1AgiUp_23 AT %MX31104.23 : BOOL;
	bSlowPull2LifterStn1AgiUp_24 AT %MX31104.24 : BOOL;
	bSlowPull2LifterStn1AgiUp_25 AT %MX31104.25 : BOOL;
	bSlowPull2LifterStn1AgiUp_26 AT %MX31104.26 : BOOL;
	bSlowPull2LifterStn1AgiUp_27 AT %MX31104.27 : BOOL;
	bSlowPull2LifterStn1AgiUp_28 AT %MX31104.28 : BOOL;
	bSlowPull2LifterStn1AgiUp_29 AT %MX31104.29 : BOOL;
	bSlowPull2LifterStn1AgiUp_30 AT %MX31104.30 : BOOL;
	bSlowPull2LifterStn1AgiUp_31 AT %MX31104.31 : BOOL;

	bSlowPull2LifterStn2AgiUp_00 AT %MX31108.0 : BOOL;
	bSlowPull2LifterStn2AgiUp_01 AT %MX31108.1 : BOOL;
	bSlowPull2LifterStn2AgiUp_02 AT %MX31108.2 : BOOL;
	bSlowPull2LifterStn2AgiUp_03 AT %MX31108.3 : BOOL;
	bSlowPull2LifterStn2AgiUp_04 AT %MX31108.4 : BOOL;
	bSlowPull2LifterStn2AgiUp_05 AT %MX31108.5 : BOOL;
	bSlowPull2LifterStn2AgiUp_06 AT %MX31108.6 : BOOL;
	bSlowPull2LifterStn2AgiUp_07 AT %MX31108.7 : BOOL;
	bSlowPull2LifterStn2AgiUp_08 AT %MX31108.8 : BOOL;
	bSlowPull2LifterStn2AgiUp_09 AT %MX31108.9 : BOOL;
	bSlowPull2LifterStn2AgiUp_10 AT %MX31108.10 : BOOL;
	bSlowPull2LifterStn2AgiUp_11 AT %MX31108.11 : BOOL;
	bSlowPull2LifterStn2AgiUp_12 AT %MX31108.12 : BOOL;
	bSlowPull2LifterStn2AgiUp_13 AT %MX31108.13 : BOOL;
	bSlowPull2LifterStn2AgiUp_14 AT %MX31108.14 : BOOL;
	bSlowPull2LifterStn2AgiUp_15 AT %MX31108.15 : BOOL;
	bSlowPull2LifterStn2AgiUp_16 AT %MX31108.16 : BOOL;
	bSlowPull2LifterStn2AgiUp_17 AT %MX31108.17 : BOOL;
	bSlowPull2LifterStn2AgiUp_18 AT %MX31108.18 : BOOL;
	bSlowPull2LifterStn2AgiUp_19 AT %MX31108.19 : BOOL;
	bSlowPull2LifterStn2AgiUp_20 AT %MX31108.20 : BOOL;
	bSlowPull2LifterStn2AgiUp_21 AT %MX31108.21 : BOOL;
	bSlowPull2LifterStn2AgiUp_22 AT %MX31108.22 : BOOL;
	bSlowPull2LifterStn2AgiUp_23 AT %MX31108.23 : BOOL;
	bSlowPull2LifterStn2AgiUp_24 AT %MX31108.24 : BOOL;
	bSlowPull2LifterStn2AgiUp_25 AT %MX31108.25 : BOOL;
	bSlowPull2LifterStn2AgiUp_26 AT %MX31108.26 : BOOL;
	bSlowPull2LifterStn2AgiUp_27 AT %MX31108.27 : BOOL;
	bSlowPull2LifterStn2AgiUp_28 AT %MX31108.28 : BOOL;
	bSlowPull2LifterStn2AgiUp_29 AT %MX31108.29 : BOOL;
	bSlowPull2LifterStn2AgiUp_30 AT %MX31108.30 : BOOL;
	bSlowPull2LifterStn2AgiUp_31 AT %MX31108.31 : BOOL;

	bSlowPull2LifterStn3AgiUp_00 AT %MX31112.0 : BOOL;
	bSlowPull2LifterStn3AgiUp_01 AT %MX31112.1 : BOOL;
	bSlowPull2LifterStn3AgiUp_02 AT %MX31112.2 : BOOL;
	bSlowPull2LifterStn3AgiUp_03 AT %MX31112.3 : BOOL;
	bSlowPull2LifterStn3AgiUp_04 AT %MX31112.4 : BOOL;
	bSlowPull2LifterStn3AgiUp_05 AT %MX31112.5 : BOOL;
	bSlowPull2LifterStn3AgiUp_06 AT %MX31112.6 : BOOL;
	bSlowPull2LifterStn3AgiUp_07 AT %MX31112.7 : BOOL;
	bSlowPull2LifterStn3AgiUp_08 AT %MX31112.8 : BOOL;
	bSlowPull2LifterStn3AgiUp_09 AT %MX31112.9 : BOOL;
	bSlowPull2LifterStn3AgiUp_10 AT %MX31112.10 : BOOL;
	bSlowPull2LifterStn3AgiUp_11 AT %MX31112.11 : BOOL;
	bSlowPull2LifterStn3AgiUp_12 AT %MX31112.12 : BOOL;
	bSlowPull2LifterStn3AgiUp_13 AT %MX31112.13 : BOOL;
	bSlowPull2LifterStn3AgiUp_14 AT %MX31112.14 : BOOL;
	bSlowPull2LifterStn3AgiUp_15 AT %MX31112.15 : BOOL;
	bSlowPull2LifterStn3AgiUp_16 AT %MX31112.16 : BOOL;
	bSlowPull2LifterStn3AgiUp_17 AT %MX31112.17 : BOOL;
	bSlowPull2LifterStn3AgiUp_18 AT %MX31112.18 : BOOL;
	bSlowPull2LifterStn3AgiUp_19 AT %MX31112.19 : BOOL;
	bSlowPull2LifterStn3AgiUp_20 AT %MX31112.20 : BOOL;
	bSlowPull2LifterStn3AgiUp_21 AT %MX31112.21 : BOOL;
	bSlowPull2LifterStn3AgiUp_22 AT %MX31112.22 : BOOL;
	bSlowPull2LifterStn3AgiUp_23 AT %MX31112.23 : BOOL;
	bSlowPull2LifterStn3AgiUp_24 AT %MX31112.24 : BOOL;
	bSlowPull2LifterStn3AgiUp_25 AT %MX31112.25 : BOOL;
	bSlowPull2LifterStn3AgiUp_26 AT %MX31112.26 : BOOL;
	bSlowPull2LifterStn3AgiUp_27 AT %MX31112.27 : BOOL;
	bSlowPull2LifterStn3AgiUp_28 AT %MX31112.28 : BOOL;
	bSlowPull2LifterStn3AgiUp_29 AT %MX31112.29 : BOOL;
	bSlowPull2LifterStn3AgiUp_30 AT %MX31112.30 : BOOL;
	bSlowPull2LifterStn3AgiUp_31 AT %MX31112.31 : BOOL;

	bSlowPull2LifterStn4AgiUp_00 AT %MX31116.0 : BOOL;
	bSlowPull2LifterStn4AgiUp_01 AT %MX31116.1 : BOOL;
	bSlowPull2LifterStn4AgiUp_02 AT %MX31116.2 : BOOL;
	bSlowPull2LifterStn4AgiUp_03 AT %MX31116.3 : BOOL;
	bSlowPull2LifterStn4AgiUp_04 AT %MX31116.4 : BOOL;
	bSlowPull2LifterStn4AgiUp_05 AT %MX31116.5 : BOOL;
	bSlowPull2LifterStn4AgiUp_06 AT %MX31116.6 : BOOL;
	bSlowPull2LifterStn4AgiUp_07 AT %MX31116.7 : BOOL;
	bSlowPull2LifterStn4AgiUp_08 AT %MX31116.8 : BOOL;
	bSlowPull2LifterStn4AgiUp_09 AT %MX31116.9 : BOOL;
	bSlowPull2LifterStn4AgiUp_10 AT %MX31116.10 : BOOL;
	bSlowPull2LifterStn4AgiUp_11 AT %MX31116.11 : BOOL;
	bSlowPull2LifterStn4AgiUp_12 AT %MX31116.12 : BOOL;
	bSlowPull2LifterStn4AgiUp_13 AT %MX31116.13 : BOOL;
	bSlowPull2LifterStn4AgiUp_14 AT %MX31116.14 : BOOL;
	bSlowPull2LifterStn4AgiUp_15 AT %MX31116.15 : BOOL;
	bSlowPull2LifterStn4AgiUp_16 AT %MX31116.16 : BOOL;
	bSlowPull2LifterStn4AgiUp_17 AT %MX31116.17 : BOOL;
	bSlowPull2LifterStn4AgiUp_18 AT %MX31116.18 : BOOL;
	bSlowPull2LifterStn4AgiUp_19 AT %MX31116.19 : BOOL;
	bSlowPull2LifterStn4AgiUp_20 AT %MX31116.20 : BOOL;
	bSlowPull2LifterStn4AgiUp_21 AT %MX31116.21 : BOOL;
	bSlowPull2LifterStn4AgiUp_22 AT %MX31116.22 : BOOL;
	bSlowPull2LifterStn4AgiUp_23 AT %MX31116.23 : BOOL;
	bSlowPull2LifterStn4AgiUp_24 AT %MX31116.24 : BOOL;
	bSlowPull2LifterStn4AgiUp_25 AT %MX31116.25 : BOOL;
	bSlowPull2LifterStn4AgiUp_26 AT %MX31116.26 : BOOL;
	bSlowPull2LifterStn4AgiUp_27 AT %MX31116.27 : BOOL;
	bSlowPull2LifterStn4AgiUp_28 AT %MX31116.28 : BOOL;
	bSlowPull2LifterStn4AgiUp_29 AT %MX31116.29 : BOOL;
	bSlowPull2LifterStn4AgiUp_30 AT %MX31116.30 : BOOL;
	bSlowPull2LifterStn4AgiUp_31 AT %MX31116.31 : BOOL;

	bSlowPull2LifterStn5AgiUp_00 AT %MX31120.0 : BOOL;
	bSlowPull2LifterStn5AgiUp_01 AT %MX31120.1 : BOOL;
	bSlowPull2LifterStn5AgiUp_02 AT %MX31120.2 : BOOL;
	bSlowPull2LifterStn5AgiUp_03 AT %MX31120.3 : BOOL;
	bSlowPull2LifterStn5AgiUp_04 AT %MX31120.4 : BOOL;
	bSlowPull2LifterStn5AgiUp_05 AT %MX31120.5 : BOOL;
	bSlowPull2LifterStn5AgiUp_06 AT %MX31120.6 : BOOL;
	bSlowPull2LifterStn5AgiUp_07 AT %MX31120.7 : BOOL;
	bSlowPull2LifterStn5AgiUp_08 AT %MX31120.8 : BOOL;
	bSlowPull2LifterStn5AgiUp_09 AT %MX31120.9 : BOOL;
	bSlowPull2LifterStn5AgiUp_10 AT %MX31120.10 : BOOL;
	bSlowPull2LifterStn5AgiUp_11 AT %MX31120.11 : BOOL;
	bSlowPull2LifterStn5AgiUp_12 AT %MX31120.12 : BOOL;
	bSlowPull2LifterStn5AgiUp_13 AT %MX31120.13 : BOOL;
	bSlowPull2LifterStn5AgiUp_14 AT %MX31120.14 : BOOL;
	bSlowPull2LifterStn5AgiUp_15 AT %MX31120.15 : BOOL;
	bSlowPull2LifterStn5AgiUp_16 AT %MX31120.16 : BOOL;
	bSlowPull2LifterStn5AgiUp_17 AT %MX31120.17 : BOOL;
	bSlowPull2LifterStn5AgiUp_18 AT %MX31120.18 : BOOL;
	bSlowPull2LifterStn5AgiUp_19 AT %MX31120.19 : BOOL;
	bSlowPull2LifterStn5AgiUp_20 AT %MX31120.20 : BOOL;
	bSlowPull2LifterStn5AgiUp_21 AT %MX31120.21 : BOOL;
	bSlowPull2LifterStn5AgiUp_22 AT %MX31120.22 : BOOL;
	bSlowPull2LifterStn5AgiUp_23 AT %MX31120.23 : BOOL;
	bSlowPull2LifterStn5AgiUp_24 AT %MX31120.24 : BOOL;
	bSlowPull2LifterStn5AgiUp_25 AT %MX31120.25 : BOOL;
	bSlowPull2LifterStn5AgiUp_26 AT %MX31120.26 : BOOL;
	bSlowPull2LifterStn5AgiUp_27 AT %MX31120.27 : BOOL;
	bSlowPull2LifterStn5AgiUp_28 AT %MX31120.28 : BOOL;
	bSlowPull2LifterStn5AgiUp_29 AT %MX31120.29 : BOOL;
	bSlowPull2LifterStn5AgiUp_30 AT %MX31120.30 : BOOL;
	bSlowPull2LifterStn5AgiUp_31 AT %MX31120.31 : BOOL;

	bSlowPull2LifterStn6AgiUp_00 AT %MX31124.0 : BOOL;
	bSlowPull2LifterStn6AgiUp_01 AT %MX31124.1 : BOOL;
	bSlowPull2LifterStn6AgiUp_02 AT %MX31124.2 : BOOL;
	bSlowPull2LifterStn6AgiUp_03 AT %MX31124.3 : BOOL;
	bSlowPull2LifterStn6AgiUp_04 AT %MX31124.4 : BOOL;
	bSlowPull2LifterStn6AgiUp_05 AT %MX31124.5 : BOOL;
	bSlowPull2LifterStn6AgiUp_06 AT %MX31124.6 : BOOL;
	bSlowPull2LifterStn6AgiUp_07 AT %MX31124.7 : BOOL;
	bSlowPull2LifterStn6AgiUp_08 AT %MX31124.8 : BOOL;
	bSlowPull2LifterStn6AgiUp_09 AT %MX31124.9 : BOOL;
	bSlowPull2LifterStn6AgiUp_10 AT %MX31124.10 : BOOL;
	bSlowPull2LifterStn6AgiUp_11 AT %MX31124.11 : BOOL;
	bSlowPull2LifterStn6AgiUp_12 AT %MX31124.12 : BOOL;
	bSlowPull2LifterStn6AgiUp_13 AT %MX31124.13 : BOOL;
	bSlowPull2LifterStn6AgiUp_14 AT %MX31124.14 : BOOL;
	bSlowPull2LifterStn6AgiUp_15 AT %MX31124.15 : BOOL;
	bSlowPull2LifterStn6AgiUp_16 AT %MX31124.16 : BOOL;
	bSlowPull2LifterStn6AgiUp_17 AT %MX31124.17 : BOOL;
	bSlowPull2LifterStn6AgiUp_18 AT %MX31124.18 : BOOL;
	bSlowPull2LifterStn6AgiUp_19 AT %MX31124.19 : BOOL;
	bSlowPull2LifterStn6AgiUp_20 AT %MX31124.20 : BOOL;
	bSlowPull2LifterStn6AgiUp_21 AT %MX31124.21 : BOOL;
	bSlowPull2LifterStn6AgiUp_22 AT %MX31124.22 : BOOL;
	bSlowPull2LifterStn6AgiUp_23 AT %MX31124.23 : BOOL;
	bSlowPull2LifterStn6AgiUp_24 AT %MX31124.24 : BOOL;
	bSlowPull2LifterStn6AgiUp_25 AT %MX31124.25 : BOOL;
	bSlowPull2LifterStn6AgiUp_26 AT %MX31124.26 : BOOL;
	bSlowPull2LifterStn6AgiUp_27 AT %MX31124.27 : BOOL;
	bSlowPull2LifterStn6AgiUp_28 AT %MX31124.28 : BOOL;
	bSlowPull2LifterStn6AgiUp_29 AT %MX31124.29 : BOOL;
	bSlowPull2LifterStn6AgiUp_30 AT %MX31124.30 : BOOL;
	bSlowPull2LifterStn6AgiUp_31 AT %MX31124.31 : BOOL;

	bSlowPull2LifterStn7AgiUp_00 AT %MX31128.0 : BOOL;
	bSlowPull2LifterStn7AgiUp_01 AT %MX31128.1 : BOOL;
	bSlowPull2LifterStn7AgiUp_02 AT %MX31128.2 : BOOL;
	bSlowPull2LifterStn7AgiUp_03 AT %MX31128.3 : BOOL;
	bSlowPull2LifterStn7AgiUp_04 AT %MX31128.4 : BOOL;
	bSlowPull2LifterStn7AgiUp_05 AT %MX31128.5 : BOOL;
	bSlowPull2LifterStn7AgiUp_06 AT %MX31128.6 : BOOL;
	bSlowPull2LifterStn7AgiUp_07 AT %MX31128.7 : BOOL;
	bSlowPull2LifterStn7AgiUp_08 AT %MX31128.8 : BOOL;
	bSlowPull2LifterStn7AgiUp_09 AT %MX31128.9 : BOOL;
	bSlowPull2LifterStn7AgiUp_10 AT %MX31128.10 : BOOL;
	bSlowPull2LifterStn7AgiUp_11 AT %MX31128.11 : BOOL;
	bSlowPull2LifterStn7AgiUp_12 AT %MX31128.12 : BOOL;
	bSlowPull2LifterStn7AgiUp_13 AT %MX31128.13 : BOOL;
	bSlowPull2LifterStn7AgiUp_14 AT %MX31128.14 : BOOL;
	bSlowPull2LifterStn7AgiUp_15 AT %MX31128.15 : BOOL;
	bSlowPull2LifterStn7AgiUp_16 AT %MX31128.16 : BOOL;
	bSlowPull2LifterStn7AgiUp_17 AT %MX31128.17 : BOOL;
	bSlowPull2LifterStn7AgiUp_18 AT %MX31128.18 : BOOL;
	bSlowPull2LifterStn7AgiUp_19 AT %MX31128.19 : BOOL;
	bSlowPull2LifterStn7AgiUp_20 AT %MX31128.20 : BOOL;
	bSlowPull2LifterStn7AgiUp_21 AT %MX31128.21 : BOOL;
	bSlowPull2LifterStn7AgiUp_22 AT %MX31128.22 : BOOL;
	bSlowPull2LifterStn7AgiUp_23 AT %MX31128.23 : BOOL;
	bSlowPull2LifterStn7AgiUp_24 AT %MX31128.24 : BOOL;
	bSlowPull2LifterStn7AgiUp_25 AT %MX31128.25 : BOOL;
	bSlowPull2LifterStn7AgiUp_26 AT %MX31128.26 : BOOL;
	bSlowPull2LifterStn7AgiUp_27 AT %MX31128.27 : BOOL;
	bSlowPull2LifterStn7AgiUp_28 AT %MX31128.28 : BOOL;
	bSlowPull2LifterStn7AgiUp_29 AT %MX31128.29 : BOOL;
	bSlowPull2LifterStn7AgiUp_30 AT %MX31128.30 : BOOL;
	bSlowPull2LifterStn7AgiUp_31 AT %MX31128.31 : BOOL;

	bSlowPull2LifterStn8AgiUp_00 AT %MX31132.0 : BOOL;
	bSlowPull2LifterStn8AgiUp_01 AT %MX31132.1 : BOOL;
	bSlowPull2LifterStn8AgiUp_02 AT %MX31132.2 : BOOL;
	bSlowPull2LifterStn8AgiUp_03 AT %MX31132.3 : BOOL;
	bSlowPull2LifterStn8AgiUp_04 AT %MX31132.4 : BOOL;
	bSlowPull2LifterStn8AgiUp_05 AT %MX31132.5 : BOOL;
	bSlowPull2LifterStn8AgiUp_06 AT %MX31132.6 : BOOL;
	bSlowPull2LifterStn8AgiUp_07 AT %MX31132.7 : BOOL;
	bSlowPull2LifterStn8AgiUp_08 AT %MX31132.8 : BOOL;
	bSlowPull2LifterStn8AgiUp_09 AT %MX31132.9 : BOOL;
	bSlowPull2LifterStn8AgiUp_10 AT %MX31132.10 : BOOL;
	bSlowPull2LifterStn8AgiUp_11 AT %MX31132.11 : BOOL;
	bSlowPull2LifterStn8AgiUp_12 AT %MX31132.12 : BOOL;
	bSlowPull2LifterStn8AgiUp_13 AT %MX31132.13 : BOOL;
	bSlowPull2LifterStn8AgiUp_14 AT %MX31132.14 : BOOL;
	bSlowPull2LifterStn8AgiUp_15 AT %MX31132.15 : BOOL;
	bSlowPull2LifterStn8AgiUp_16 AT %MX31132.16 : BOOL;
	bSlowPull2LifterStn8AgiUp_17 AT %MX31132.17 : BOOL;
	bSlowPull2LifterStn8AgiUp_18 AT %MX31132.18 : BOOL;
	bSlowPull2LifterStn8AgiUp_19 AT %MX31132.19 : BOOL;
	bSlowPull2LifterStn8AgiUp_20 AT %MX31132.20 : BOOL;
	bSlowPull2LifterStn8AgiUp_21 AT %MX31132.21 : BOOL;
	bSlowPull2LifterStn8AgiUp_22 AT %MX31132.22 : BOOL;
	bSlowPull2LifterStn8AgiUp_23 AT %MX31132.23 : BOOL;
	bSlowPull2LifterStn8AgiUp_24 AT %MX31132.24 : BOOL;
	bSlowPull2LifterStn8AgiUp_25 AT %MX31132.25 : BOOL;
	bSlowPull2LifterStn8AgiUp_26 AT %MX31132.26 : BOOL;
	bSlowPull2LifterStn8AgiUp_27 AT %MX31132.27 : BOOL;
	bSlowPull2LifterStn8AgiUp_28 AT %MX31132.28 : BOOL;
	bSlowPull2LifterStn8AgiUp_29 AT %MX31132.29 : BOOL;
	bSlowPull2LifterStn8AgiUp_30 AT %MX31132.30 : BOOL;
	bSlowPull2LifterStn8AgiUp_31 AT %MX31132.31 : BOOL;

	bSlowPull2LifterStn9AgiUp_00 AT %MX31136.0 : BOOL;
	bSlowPull2LifterStn9AgiUp_01 AT %MX31136.1 : BOOL;
	bSlowPull2LifterStn9AgiUp_02 AT %MX31136.2 : BOOL;
	bSlowPull2LifterStn9AgiUp_03 AT %MX31136.3 : BOOL;
	bSlowPull2LifterStn9AgiUp_04 AT %MX31136.4 : BOOL;
	bSlowPull2LifterStn9AgiUp_05 AT %MX31136.5 : BOOL;
	bSlowPull2LifterStn9AgiUp_06 AT %MX31136.6 : BOOL;
	bSlowPull2LifterStn9AgiUp_07 AT %MX31136.7 : BOOL;
	bSlowPull2LifterStn9AgiUp_08 AT %MX31136.8 : BOOL;
	bSlowPull2LifterStn9AgiUp_09 AT %MX31136.9 : BOOL;
	bSlowPull2LifterStn9AgiUp_10 AT %MX31136.10 : BOOL;
	bSlowPull2LifterStn9AgiUp_11 AT %MX31136.11 : BOOL;
	bSlowPull2LifterStn9AgiUp_12 AT %MX31136.12 : BOOL;
	bSlowPull2LifterStn9AgiUp_13 AT %MX31136.13 : BOOL;
	bSlowPull2LifterStn9AgiUp_14 AT %MX31136.14 : BOOL;
	bSlowPull2LifterStn9AgiUp_15 AT %MX31136.15 : BOOL;
	bSlowPull2LifterStn9AgiUp_16 AT %MX31136.16 : BOOL;
	bSlowPull2LifterStn9AgiUp_17 AT %MX31136.17 : BOOL;
	bSlowPull2LifterStn9AgiUp_18 AT %MX31136.18 : BOOL;
	bSlowPull2LifterStn9AgiUp_19 AT %MX31136.19 : BOOL;
	bSlowPull2LifterStn9AgiUp_20 AT %MX31136.20 : BOOL;
	bSlowPull2LifterStn9AgiUp_21 AT %MX31136.21 : BOOL;
	bSlowPull2LifterStn9AgiUp_22 AT %MX31136.22 : BOOL;
	bSlowPull2LifterStn9AgiUp_23 AT %MX31136.23 : BOOL;
	bSlowPull2LifterStn9AgiUp_24 AT %MX31136.24 : BOOL;
	bSlowPull2LifterStn9AgiUp_25 AT %MX31136.25 : BOOL;
	bSlowPull2LifterStn9AgiUp_26 AT %MX31136.26 : BOOL;
	bSlowPull2LifterStn9AgiUp_27 AT %MX31136.27 : BOOL;
	bSlowPull2LifterStn9AgiUp_28 AT %MX31136.28 : BOOL;
	bSlowPull2LifterStn9AgiUp_29 AT %MX31136.29 : BOOL;
	bSlowPull2LifterStn9AgiUp_30 AT %MX31136.30 : BOOL;
	bSlowPull2LifterStn9AgiUp_31 AT %MX31136.31 : BOOL;

	bSlowPull2LifterStn10AgiUp_00 AT %MX31140.0 : BOOL;
	bSlowPull2LifterStn10AgiUp_01 AT %MX31140.1 : BOOL;
	bSlowPull2LifterStn10AgiUp_02 AT %MX31140.2 : BOOL;
	bSlowPull2LifterStn10AgiUp_03 AT %MX31140.3 : BOOL;
	bSlowPull2LifterStn10AgiUp_04 AT %MX31140.4 : BOOL;
	bSlowPull2LifterStn10AgiUp_05 AT %MX31140.5 : BOOL;
	bSlowPull2LifterStn10AgiUp_06 AT %MX31140.6 : BOOL;
	bSlowPull2LifterStn10AgiUp_07 AT %MX31140.7 : BOOL;
	bSlowPull2LifterStn10AgiUp_08 AT %MX31140.8 : BOOL;
	bSlowPull2LifterStn10AgiUp_09 AT %MX31140.9 : BOOL;
	bSlowPull2LifterStn10AgiUp_10 AT %MX31140.10 : BOOL;
	bSlowPull2LifterStn10AgiUp_11 AT %MX31140.11 : BOOL;
	bSlowPull2LifterStn10AgiUp_12 AT %MX31140.12 : BOOL;
	bSlowPull2LifterStn10AgiUp_13 AT %MX31140.13 : BOOL;
	bSlowPull2LifterStn10AgiUp_14 AT %MX31140.14 : BOOL;
	bSlowPull2LifterStn10AgiUp_15 AT %MX31140.15 : BOOL;
	bSlowPull2LifterStn10AgiUp_16 AT %MX31140.16 : BOOL;
	bSlowPull2LifterStn10AgiUp_17 AT %MX31140.17 : BOOL;
	bSlowPull2LifterStn10AgiUp_18 AT %MX31140.18 : BOOL;
	bSlowPull2LifterStn10AgiUp_19 AT %MX31140.19 : BOOL;
	bSlowPull2LifterStn10AgiUp_20 AT %MX31140.20 : BOOL;
	bSlowPull2LifterStn10AgiUp_21 AT %MX31140.21 : BOOL;
	bSlowPull2LifterStn10AgiUp_22 AT %MX31140.22 : BOOL;
	bSlowPull2LifterStn10AgiUp_23 AT %MX31140.23 : BOOL;
	bSlowPull2LifterStn10AgiUp_24 AT %MX31140.24 : BOOL;
	bSlowPull2LifterStn10AgiUp_25 AT %MX31140.25 : BOOL;
	bSlowPull2LifterStn10AgiUp_26 AT %MX31140.26 : BOOL;
	bSlowPull2LifterStn10AgiUp_27 AT %MX31140.27 : BOOL;
	bSlowPull2LifterStn10AgiUp_28 AT %MX31140.28 : BOOL;
	bSlowPull2LifterStn10AgiUp_29 AT %MX31140.29 : BOOL;
	bSlowPull2LifterStn10AgiUp_30 AT %MX31140.30 : BOOL;
	bSlowPull2LifterStn10AgiUp_31 AT %MX31140.31 : BOOL;

	bSlowPull2LifterStn11AgiUp_00 AT %MX31144.0 : BOOL;
	bSlowPull2LifterStn11AgiUp_01 AT %MX31144.1 : BOOL;
	bSlowPull2LifterStn11AgiUp_02 AT %MX31144.2 : BOOL;
	bSlowPull2LifterStn11AgiUp_03 AT %MX31144.3 : BOOL;
	bSlowPull2LifterStn11AgiUp_04 AT %MX31144.4 : BOOL;
	bSlowPull2LifterStn11AgiUp_05 AT %MX31144.5 : BOOL;
	bSlowPull2LifterStn11AgiUp_06 AT %MX31144.6 : BOOL;
	bSlowPull2LifterStn11AgiUp_07 AT %MX31144.7 : BOOL;
	bSlowPull2LifterStn11AgiUp_08 AT %MX31144.8 : BOOL;
	bSlowPull2LifterStn11AgiUp_09 AT %MX31144.9 : BOOL;
	bSlowPull2LifterStn11AgiUp_10 AT %MX31144.10 : BOOL;
	bSlowPull2LifterStn11AgiUp_11 AT %MX31144.11 : BOOL;
	bSlowPull2LifterStn11AgiUp_12 AT %MX31144.12 : BOOL;
	bSlowPull2LifterStn11AgiUp_13 AT %MX31144.13 : BOOL;
	bSlowPull2LifterStn11AgiUp_14 AT %MX31144.14 : BOOL;
	bSlowPull2LifterStn11AgiUp_15 AT %MX31144.15 : BOOL;
	bSlowPull2LifterStn11AgiUp_16 AT %MX31144.16 : BOOL;
	bSlowPull2LifterStn11AgiUp_17 AT %MX31144.17 : BOOL;
	bSlowPull2LifterStn11AgiUp_18 AT %MX31144.18 : BOOL;
	bSlowPull2LifterStn11AgiUp_19 AT %MX31144.19 : BOOL;
	bSlowPull2LifterStn11AgiUp_20 AT %MX31144.20 : BOOL;
	bSlowPull2LifterStn11AgiUp_21 AT %MX31144.21 : BOOL;
	bSlowPull2LifterStn11AgiUp_22 AT %MX31144.22 : BOOL;
	bSlowPull2LifterStn11AgiUp_23 AT %MX31144.23 : BOOL;
	bSlowPull2LifterStn11AgiUp_24 AT %MX31144.24 : BOOL;
	bSlowPull2LifterStn11AgiUp_25 AT %MX31144.25 : BOOL;
	bSlowPull2LifterStn11AgiUp_26 AT %MX31144.26 : BOOL;
	bSlowPull2LifterStn11AgiUp_27 AT %MX31144.27 : BOOL;
	bSlowPull2LifterStn11AgiUp_28 AT %MX31144.28 : BOOL;
	bSlowPull2LifterStn11AgiUp_29 AT %MX31144.29 : BOOL;
	bSlowPull2LifterStn11AgiUp_30 AT %MX31144.30 : BOOL;
	bSlowPull2LifterStn11AgiUp_31 AT %MX31144.31 : BOOL;

	bSlowPull2LifterStn12AgiUp_00 AT %MX31148.0 : BOOL;
	bSlowPull2LifterStn12AgiUp_01 AT %MX31148.1 : BOOL;
	bSlowPull2LifterStn12AgiUp_02 AT %MX31148.2 : BOOL;
	bSlowPull2LifterStn12AgiUp_03 AT %MX31148.3 : BOOL;
	bSlowPull2LifterStn12AgiUp_04 AT %MX31148.4 : BOOL;
	bSlowPull2LifterStn12AgiUp_05 AT %MX31148.5 : BOOL;
	bSlowPull2LifterStn12AgiUp_06 AT %MX31148.6 : BOOL;
	bSlowPull2LifterStn12AgiUp_07 AT %MX31148.7 : BOOL;
	bSlowPull2LifterStn12AgiUp_08 AT %MX31148.8 : BOOL;
	bSlowPull2LifterStn12AgiUp_09 AT %MX31148.9 : BOOL;
	bSlowPull2LifterStn12AgiUp_10 AT %MX31148.10 : BOOL;
	bSlowPull2LifterStn12AgiUp_11 AT %MX31148.11 : BOOL;
	bSlowPull2LifterStn12AgiUp_12 AT %MX31148.12 : BOOL;
	bSlowPull2LifterStn12AgiUp_13 AT %MX31148.13 : BOOL;
	bSlowPull2LifterStn12AgiUp_14 AT %MX31148.14 : BOOL;
	bSlowPull2LifterStn12AgiUp_15 AT %MX31148.15 : BOOL;
	bSlowPull2LifterStn12AgiUp_16 AT %MX31148.16 : BOOL;
	bSlowPull2LifterStn12AgiUp_17 AT %MX31148.17 : BOOL;
	bSlowPull2LifterStn12AgiUp_18 AT %MX31148.18 : BOOL;
	bSlowPull2LifterStn12AgiUp_19 AT %MX31148.19 : BOOL;
	bSlowPull2LifterStn12AgiUp_20 AT %MX31148.20 : BOOL;
	bSlowPull2LifterStn12AgiUp_21 AT %MX31148.21 : BOOL;
	bSlowPull2LifterStn12AgiUp_22 AT %MX31148.22 : BOOL;
	bSlowPull2LifterStn12AgiUp_23 AT %MX31148.23 : BOOL;
	bSlowPull2LifterStn12AgiUp_24 AT %MX31148.24 : BOOL;
	bSlowPull2LifterStn12AgiUp_25 AT %MX31148.25 : BOOL;
	bSlowPull2LifterStn12AgiUp_26 AT %MX31148.26 : BOOL;
	bSlowPull2LifterStn12AgiUp_27 AT %MX31148.27 : BOOL;
	bSlowPull2LifterStn12AgiUp_28 AT %MX31148.28 : BOOL;
	bSlowPull2LifterStn12AgiUp_29 AT %MX31148.29 : BOOL;
	bSlowPull2LifterStn12AgiUp_30 AT %MX31148.30 : BOOL;
	bSlowPull2LifterStn12AgiUp_31 AT %MX31148.31 : BOOL;


(* xxxxxxxxxxxxxxxxxxxxxxxxxxxxxxxxxxxxxxx Lifter xxxxxxxxxxxxxxxxxxxxxxxxxxxxxxxxxxxxxxx*)
(*========= Up/Down LifterAgiDown BOOL LINK with %MX31000-  =========*)

	bSlowPull2LifterStn1AgiDown_00 AT %MX31204.0 : BOOL;
	bSlowPull2LifterStn1AgiDown_01 AT %MX31204.1 : BOOL;
	bSlowPull2LifterStn1AgiDown_02 AT %MX31204.2 : BOOL;
	bSlowPull2LifterStn1AgiDown_03 AT %MX31204.3 : BOOL;
	bSlowPull2LifterStn1AgiDown_04 AT %MX31204.4 : BOOL;
	bSlowPull2LifterStn1AgiDown_05 AT %MX31204.5 : BOOL;
	bSlowPull2LifterStn1AgiDown_06 AT %MX31204.6 : BOOL;
	bSlowPull2LifterStn1AgiDown_07 AT %MX31204.7 : BOOL;
	bSlowPull2LifterStn1AgiDown_08 AT %MX31204.8 : BOOL;
	bSlowPull2LifterStn1AgiDown_09 AT %MX31204.9 : BOOL;
	bSlowPull2LifterStn1AgiDown_10 AT %MX31204.10 : BOOL;
	bSlowPull2LifterStn1AgiDown_11 AT %MX31204.11 : BOOL;
	bSlowPull2LifterStn1AgiDown_12 AT %MX31204.12 : BOOL;
	bSlowPull2LifterStn1AgiDown_13 AT %MX31204.13 : BOOL;
	bSlowPull2LifterStn1AgiDown_14 AT %MX31204.14 : BOOL;
	bSlowPull2LifterStn1AgiDown_15 AT %MX31204.15 : BOOL;
	bSlowPull2LifterStn1AgiDown_16 AT %MX31204.16 : BOOL;
	bSlowPull2LifterStn1AgiDown_17 AT %MX31204.17 : BOOL;
	bSlowPull2LifterStn1AgiDown_18 AT %MX31204.18 : BOOL;
	bSlowPull2LifterStn1AgiDown_19 AT %MX31204.19 : BOOL;
	bSlowPull2LifterStn1AgiDown_20 AT %MX31204.20 : BOOL;
	bSlowPull2LifterStn1AgiDown_21 AT %MX31204.21 : BOOL;
	bSlowPull2LifterStn1AgiDown_22 AT %MX31204.22 : BOOL;
	bSlowPull2LifterStn1AgiDown_23 AT %MX31204.23 : BOOL;
	bSlowPull2LifterStn1AgiDown_24 AT %MX31204.24 : BOOL;
	bSlowPull2LifterStn1AgiDown_25 AT %MX31204.25 : BOOL;
	bSlowPull2LifterStn1AgiDown_26 AT %MX31204.26 : BOOL;
	bSlowPull2LifterStn1AgiDown_27 AT %MX31204.27 : BOOL;
	bSlowPull2LifterStn1AgiDown_28 AT %MX31204.28 : BOOL;
	bSlowPull2LifterStn1AgiDown_29 AT %MX31204.29 : BOOL;
	bSlowPull2LifterStn1AgiDown_30 AT %MX31204.30 : BOOL;
	bSlowPull2LifterStn1AgiDown_31 AT %MX31204.31 : BOOL;

	bSlowPull2LifterStn2AgiDown_00 AT %MX31208.0 : BOOL;
	bSlowPull2LifterStn2AgiDown_01 AT %MX31208.1 : BOOL;
	bSlowPull2LifterStn2AgiDown_02 AT %MX31208.2 : BOOL;
	bSlowPull2LifterStn2AgiDown_03 AT %MX31208.3 : BOOL;
	bSlowPull2LifterStn2AgiDown_04 AT %MX31208.4 : BOOL;
	bSlowPull2LifterStn2AgiDown_05 AT %MX31208.5 : BOOL;
	bSlowPull2LifterStn2AgiDown_06 AT %MX31208.6 : BOOL;
	bSlowPull2LifterStn2AgiDown_07 AT %MX31208.7 : BOOL;
	bSlowPull2LifterStn2AgiDown_08 AT %MX31208.8 : BOOL;
	bSlowPull2LifterStn2AgiDown_09 AT %MX31208.9 : BOOL;
	bSlowPull2LifterStn2AgiDown_10 AT %MX31208.10 : BOOL;
	bSlowPull2LifterStn2AgiDown_11 AT %MX31208.11 : BOOL;
	bSlowPull2LifterStn2AgiDown_12 AT %MX31208.12 : BOOL;
	bSlowPull2LifterStn2AgiDown_13 AT %MX31208.13 : BOOL;
	bSlowPull2LifterStn2AgiDown_14 AT %MX31208.14 : BOOL;
	bSlowPull2LifterStn2AgiDown_15 AT %MX31208.15 : BOOL;
	bSlowPull2LifterStn2AgiDown_16 AT %MX31208.16 : BOOL;
	bSlowPull2LifterStn2AgiDown_17 AT %MX31208.17 : BOOL;
	bSlowPull2LifterStn2AgiDown_18 AT %MX31208.18 : BOOL;
	bSlowPull2LifterStn2AgiDown_19 AT %MX31208.19 : BOOL;
	bSlowPull2LifterStn2AgiDown_20 AT %MX31208.20 : BOOL;
	bSlowPull2LifterStn2AgiDown_21 AT %MX31208.21 : BOOL;
	bSlowPull2LifterStn2AgiDown_22 AT %MX31208.22 : BOOL;
	bSlowPull2LifterStn2AgiDown_23 AT %MX31208.23 : BOOL;
	bSlowPull2LifterStn2AgiDown_24 AT %MX31208.24 : BOOL;
	bSlowPull2LifterStn2AgiDown_25 AT %MX31208.25 : BOOL;
	bSlowPull2LifterStn2AgiDown_26 AT %MX31208.26 : BOOL;
	bSlowPull2LifterStn2AgiDown_27 AT %MX31208.27 : BOOL;
	bSlowPull2LifterStn2AgiDown_28 AT %MX31208.28 : BOOL;
	bSlowPull2LifterStn2AgiDown_29 AT %MX31208.29 : BOOL;
	bSlowPull2LifterStn2AgiDown_30 AT %MX31208.30 : BOOL;
	bSlowPull2LifterStn2AgiDown_31 AT %MX31208.31 : BOOL;

	bSlowPull2LifterStn3AgiDown_00 AT %MX31212.0 : BOOL;
	bSlowPull2LifterStn3AgiDown_01 AT %MX31212.1 : BOOL;
	bSlowPull2LifterStn3AgiDown_02 AT %MX31212.2 : BOOL;
	bSlowPull2LifterStn3AgiDown_03 AT %MX31212.3 : BOOL;
	bSlowPull2LifterStn3AgiDown_04 AT %MX31212.4 : BOOL;
	bSlowPull2LifterStn3AgiDown_05 AT %MX31212.5 : BOOL;
	bSlowPull2LifterStn3AgiDown_06 AT %MX31212.6 : BOOL;
	bSlowPull2LifterStn3AgiDown_07 AT %MX31212.7 : BOOL;
	bSlowPull2LifterStn3AgiDown_08 AT %MX31212.8 : BOOL;
	bSlowPull2LifterStn3AgiDown_09 AT %MX31212.9 : BOOL;
	bSlowPull2LifterStn3AgiDown_10 AT %MX31212.10 : BOOL;
	bSlowPull2LifterStn3AgiDown_11 AT %MX31212.11 : BOOL;
	bSlowPull2LifterStn3AgiDown_12 AT %MX31212.12 : BOOL;
	bSlowPull2LifterStn3AgiDown_13 AT %MX31212.13 : BOOL;
	bSlowPull2LifterStn3AgiDown_14 AT %MX31212.14 : BOOL;
	bSlowPull2LifterStn3AgiDown_15 AT %MX31212.15 : BOOL;
	bSlowPull2LifterStn3AgiDown_16 AT %MX31212.16 : BOOL;
	bSlowPull2LifterStn3AgiDown_17 AT %MX31212.17 : BOOL;
	bSlowPull2LifterStn3AgiDown_18 AT %MX31212.18 : BOOL;
	bSlowPull2LifterStn3AgiDown_19 AT %MX31212.19 : BOOL;
	bSlowPull2LifterStn3AgiDown_20 AT %MX31212.20 : BOOL;
	bSlowPull2LifterStn3AgiDown_21 AT %MX31212.21 : BOOL;
	bSlowPull2LifterStn3AgiDown_22 AT %MX31212.22 : BOOL;
	bSlowPull2LifterStn3AgiDown_23 AT %MX31212.23 : BOOL;
	bSlowPull2LifterStn3AgiDown_24 AT %MX31212.24 : BOOL;
	bSlowPull2LifterStn3AgiDown_25 AT %MX31212.25 : BOOL;
	bSlowPull2LifterStn3AgiDown_26 AT %MX31212.26 : BOOL;
	bSlowPull2LifterStn3AgiDown_27 AT %MX31212.27 : BOOL;
	bSlowPull2LifterStn3AgiDown_28 AT %MX31212.28 : BOOL;
	bSlowPull2LifterStn3AgiDown_29 AT %MX31212.29 : BOOL;
	bSlowPull2LifterStn3AgiDown_30 AT %MX31212.30 : BOOL;
	bSlowPull2LifterStn3AgiDown_31 AT %MX31212.31 : BOOL;

	bSlowPull2LifterStn4AgiDown_00 AT %MX31216.0 : BOOL;
	bSlowPull2LifterStn4AgiDown_01 AT %MX31216.1 : BOOL;
	bSlowPull2LifterStn4AgiDown_02 AT %MX31216.2 : BOOL;
	bSlowPull2LifterStn4AgiDown_03 AT %MX31216.3 : BOOL;
	bSlowPull2LifterStn4AgiDown_04 AT %MX31216.4 : BOOL;
	bSlowPull2LifterStn4AgiDown_05 AT %MX31216.5 : BOOL;
	bSlowPull2LifterStn4AgiDown_06 AT %MX31216.6 : BOOL;
	bSlowPull2LifterStn4AgiDown_07 AT %MX31216.7 : BOOL;
	bSlowPull2LifterStn4AgiDown_08 AT %MX31216.8 : BOOL;
	bSlowPull2LifterStn4AgiDown_09 AT %MX31216.9 : BOOL;
	bSlowPull2LifterStn4AgiDown_10 AT %MX31216.10 : BOOL;
	bSlowPull2LifterStn4AgiDown_11 AT %MX31216.11 : BOOL;
	bSlowPull2LifterStn4AgiDown_12 AT %MX31216.12 : BOOL;
	bSlowPull2LifterStn4AgiDown_13 AT %MX31216.13 : BOOL;
	bSlowPull2LifterStn4AgiDown_14 AT %MX31216.14 : BOOL;
	bSlowPull2LifterStn4AgiDown_15 AT %MX31216.15 : BOOL;
	bSlowPull2LifterStn4AgiDown_16 AT %MX31216.16 : BOOL;
	bSlowPull2LifterStn4AgiDown_17 AT %MX31216.17 : BOOL;
	bSlowPull2LifterStn4AgiDown_18 AT %MX31216.18 : BOOL;
	bSlowPull2LifterStn4AgiDown_19 AT %MX31216.19 : BOOL;
	bSlowPull2LifterStn4AgiDown_20 AT %MX31216.20 : BOOL;
	bSlowPull2LifterStn4AgiDown_21 AT %MX31216.21 : BOOL;
	bSlowPull2LifterStn4AgiDown_22 AT %MX31216.22 : BOOL;
	bSlowPull2LifterStn4AgiDown_23 AT %MX31216.23 : BOOL;
	bSlowPull2LifterStn4AgiDown_24 AT %MX31216.24 : BOOL;
	bSlowPull2LifterStn4AgiDown_25 AT %MX31216.25 : BOOL;
	bSlowPull2LifterStn4AgiDown_26 AT %MX31216.26 : BOOL;
	bSlowPull2LifterStn4AgiDown_27 AT %MX31216.27 : BOOL;
	bSlowPull2LifterStn4AgiDown_28 AT %MX31216.28 : BOOL;
	bSlowPull2LifterStn4AgiDown_29 AT %MX31216.29 : BOOL;
	bSlowPull2LifterStn4AgiDown_30 AT %MX31216.30 : BOOL;
	bSlowPull2LifterStn4AgiDown_31 AT %MX31216.31 : BOOL;

	bSlowPull2LifterStn5AgiDown_00 AT %MX31220.0 : BOOL;
	bSlowPull2LifterStn5AgiDown_01 AT %MX31220.1 : BOOL;
	bSlowPull2LifterStn5AgiDown_02 AT %MX31220.2 : BOOL;
	bSlowPull2LifterStn5AgiDown_03 AT %MX31220.3 : BOOL;
	bSlowPull2LifterStn5AgiDown_04 AT %MX31220.4 : BOOL;
	bSlowPull2LifterStn5AgiDown_05 AT %MX31220.5 : BOOL;
	bSlowPull2LifterStn5AgiDown_06 AT %MX31220.6 : BOOL;
	bSlowPull2LifterStn5AgiDown_07 AT %MX31220.7 : BOOL;
	bSlowPull2LifterStn5AgiDown_08 AT %MX31220.8 : BOOL;
	bSlowPull2LifterStn5AgiDown_09 AT %MX31220.9 : BOOL;
	bSlowPull2LifterStn5AgiDown_10 AT %MX31220.10 : BOOL;
	bSlowPull2LifterStn5AgiDown_11 AT %MX31220.11 : BOOL;
	bSlowPull2LifterStn5AgiDown_12 AT %MX31220.12 : BOOL;
	bSlowPull2LifterStn5AgiDown_13 AT %MX31220.13 : BOOL;
	bSlowPull2LifterStn5AgiDown_14 AT %MX31220.14 : BOOL;
	bSlowPull2LifterStn5AgiDown_15 AT %MX31220.15 : BOOL;
	bSlowPull2LifterStn5AgiDown_16 AT %MX31220.16 : BOOL;
	bSlowPull2LifterStn5AgiDown_17 AT %MX31220.17 : BOOL;
	bSlowPull2LifterStn5AgiDown_18 AT %MX31220.18 : BOOL;
	bSlowPull2LifterStn5AgiDown_19 AT %MX31220.19 : BOOL;
	bSlowPull2LifterStn5AgiDown_20 AT %MX31220.20 : BOOL;
	bSlowPull2LifterStn5AgiDown_21 AT %MX31220.21 : BOOL;
	bSlowPull2LifterStn5AgiDown_22 AT %MX31220.22 : BOOL;
	bSlowPull2LifterStn5AgiDown_23 AT %MX31220.23 : BOOL;
	bSlowPull2LifterStn5AgiDown_24 AT %MX31220.24 : BOOL;
	bSlowPull2LifterStn5AgiDown_25 AT %MX31220.25 : BOOL;
	bSlowPull2LifterStn5AgiDown_26 AT %MX31220.26 : BOOL;
	bSlowPull2LifterStn5AgiDown_27 AT %MX31220.27 : BOOL;
	bSlowPull2LifterStn5AgiDown_28 AT %MX31220.28 : BOOL;
	bSlowPull2LifterStn5AgiDown_29 AT %MX31220.29 : BOOL;
	bSlowPull2LifterStn5AgiDown_30 AT %MX31220.30 : BOOL;
	bSlowPull2LifterStn5AgiDown_31 AT %MX31220.31 : BOOL;

	bSlowPull2LifterStn6AgiDown_00 AT %MX31224.0 : BOOL;
	bSlowPull2LifterStn6AgiDown_01 AT %MX31224.1 : BOOL;
	bSlowPull2LifterStn6AgiDown_02 AT %MX31224.2 : BOOL;
	bSlowPull2LifterStn6AgiDown_03 AT %MX31224.3 : BOOL;
	bSlowPull2LifterStn6AgiDown_04 AT %MX31224.4 : BOOL;
	bSlowPull2LifterStn6AgiDown_05 AT %MX31224.5 : BOOL;
	bSlowPull2LifterStn6AgiDown_06 AT %MX31224.6 : BOOL;
	bSlowPull2LifterStn6AgiDown_07 AT %MX31224.7 : BOOL;
	bSlowPull2LifterStn6AgiDown_08 AT %MX31224.8 : BOOL;
	bSlowPull2LifterStn6AgiDown_09 AT %MX31224.9 : BOOL;
	bSlowPull2LifterStn6AgiDown_10 AT %MX31224.10 : BOOL;
	bSlowPull2LifterStn6AgiDown_11 AT %MX31224.11 : BOOL;
	bSlowPull2LifterStn6AgiDown_12 AT %MX31224.12 : BOOL;
	bSlowPull2LifterStn6AgiDown_13 AT %MX31224.13 : BOOL;
	bSlowPull2LifterStn6AgiDown_14 AT %MX31224.14 : BOOL;
	bSlowPull2LifterStn6AgiDown_15 AT %MX31224.15 : BOOL;
	bSlowPull2LifterStn6AgiDown_16 AT %MX31224.16 : BOOL;
	bSlowPull2LifterStn6AgiDown_17 AT %MX31224.17 : BOOL;
	bSlowPull2LifterStn6AgiDown_18 AT %MX31224.18 : BOOL;
	bSlowPull2LifterStn6AgiDown_19 AT %MX31224.19 : BOOL;
	bSlowPull2LifterStn6AgiDown_20 AT %MX31224.20 : BOOL;
	bSlowPull2LifterStn6AgiDown_21 AT %MX31224.21 : BOOL;
	bSlowPull2LifterStn6AgiDown_22 AT %MX31224.22 : BOOL;
	bSlowPull2LifterStn6AgiDown_23 AT %MX31224.23 : BOOL;
	bSlowPull2LifterStn6AgiDown_24 AT %MX31224.24 : BOOL;
	bSlowPull2LifterStn6AgiDown_25 AT %MX31224.25 : BOOL;
	bSlowPull2LifterStn6AgiDown_26 AT %MX31224.26 : BOOL;
	bSlowPull2LifterStn6AgiDown_27 AT %MX31224.27 : BOOL;
	bSlowPull2LifterStn6AgiDown_28 AT %MX31224.28 : BOOL;
	bSlowPull2LifterStn6AgiDown_29 AT %MX31224.29 : BOOL;
	bSlowPull2LifterStn6AgiDown_30 AT %MX31224.30 : BOOL;
	bSlowPull2LifterStn6AgiDown_31 AT %MX31224.31 : BOOL;

	bSlowPull2LifterStn7AgiDown_00 AT %MX31228.0 : BOOL;
	bSlowPull2LifterStn7AgiDown_01 AT %MX31228.1 : BOOL;
	bSlowPull2LifterStn7AgiDown_02 AT %MX31228.2 : BOOL;
	bSlowPull2LifterStn7AgiDown_03 AT %MX31228.3 : BOOL;
	bSlowPull2LifterStn7AgiDown_04 AT %MX31228.4 : BOOL;
	bSlowPull2LifterStn7AgiDown_05 AT %MX31228.5 : BOOL;
	bSlowPull2LifterStn7AgiDown_06 AT %MX31228.6 : BOOL;
	bSlowPull2LifterStn7AgiDown_07 AT %MX31228.7 : BOOL;
	bSlowPull2LifterStn7AgiDown_08 AT %MX31228.8 : BOOL;
	bSlowPull2LifterStn7AgiDown_09 AT %MX31228.9 : BOOL;
	bSlowPull2LifterStn7AgiDown_10 AT %MX31228.10 : BOOL;
	bSlowPull2LifterStn7AgiDown_11 AT %MX31228.11 : BOOL;
	bSlowPull2LifterStn7AgiDown_12 AT %MX31228.12 : BOOL;
	bSlowPull2LifterStn7AgiDown_13 AT %MX31228.13 : BOOL;
	bSlowPull2LifterStn7AgiDown_14 AT %MX31228.14 : BOOL;
	bSlowPull2LifterStn7AgiDown_15 AT %MX31228.15 : BOOL;
	bSlowPull2LifterStn7AgiDown_16 AT %MX31228.16 : BOOL;
	bSlowPull2LifterStn7AgiDown_17 AT %MX31228.17 : BOOL;
	bSlowPull2LifterStn7AgiDown_18 AT %MX31228.18 : BOOL;
	bSlowPull2LifterStn7AgiDown_19 AT %MX31228.19 : BOOL;
	bSlowPull2LifterStn7AgiDown_20 AT %MX31228.20 : BOOL;
	bSlowPull2LifterStn7AgiDown_21 AT %MX31228.21 : BOOL;
	bSlowPull2LifterStn7AgiDown_22 AT %MX31228.22 : BOOL;
	bSlowPull2LifterStn7AgiDown_23 AT %MX31228.23 : BOOL;
	bSlowPull2LifterStn7AgiDown_24 AT %MX31228.24 : BOOL;
	bSlowPull2LifterStn7AgiDown_25 AT %MX31228.25 : BOOL;
	bSlowPull2LifterStn7AgiDown_26 AT %MX31228.26 : BOOL;
	bSlowPull2LifterStn7AgiDown_27 AT %MX31228.27 : BOOL;
	bSlowPull2LifterStn7AgiDown_28 AT %MX31228.28 : BOOL;
	bSlowPull2LifterStn7AgiDown_29 AT %MX31228.29 : BOOL;
	bSlowPull2LifterStn7AgiDown_30 AT %MX31228.30 : BOOL;
	bSlowPull2LifterStn7AgiDown_31 AT %MX31228.31 : BOOL;

	bSlowPull2LifterStn8AgiDown_00 AT %MX31232.0 : BOOL;
	bSlowPull2LifterStn8AgiDown_01 AT %MX31232.1 : BOOL;
	bSlowPull2LifterStn8AgiDown_02 AT %MX31232.2 : BOOL;
	bSlowPull2LifterStn8AgiDown_03 AT %MX31232.3 : BOOL;
	bSlowPull2LifterStn8AgiDown_04 AT %MX31232.4 : BOOL;
	bSlowPull2LifterStn8AgiDown_05 AT %MX31232.5 : BOOL;
	bSlowPull2LifterStn8AgiDown_06 AT %MX31232.6 : BOOL;
	bSlowPull2LifterStn8AgiDown_07 AT %MX31232.7 : BOOL;
	bSlowPull2LifterStn8AgiDown_08 AT %MX31232.8 : BOOL;
	bSlowPull2LifterStn8AgiDown_09 AT %MX31232.9 : BOOL;
	bSlowPull2LifterStn8AgiDown_10 AT %MX31232.10 : BOOL;
	bSlowPull2LifterStn8AgiDown_11 AT %MX31232.11 : BOOL;
	bSlowPull2LifterStn8AgiDown_12 AT %MX31232.12 : BOOL;
	bSlowPull2LifterStn8AgiDown_13 AT %MX31232.13 : BOOL;
	bSlowPull2LifterStn8AgiDown_14 AT %MX31232.14 : BOOL;
	bSlowPull2LifterStn8AgiDown_15 AT %MX31232.15 : BOOL;
	bSlowPull2LifterStn8AgiDown_16 AT %MX31232.16 : BOOL;
	bSlowPull2LifterStn8AgiDown_17 AT %MX31232.17 : BOOL;
	bSlowPull2LifterStn8AgiDown_18 AT %MX31232.18 : BOOL;
	bSlowPull2LifterStn8AgiDown_19 AT %MX31232.19 : BOOL;
	bSlowPull2LifterStn8AgiDown_20 AT %MX31232.20 : BOOL;
	bSlowPull2LifterStn8AgiDown_21 AT %MX31232.21 : BOOL;
	bSlowPull2LifterStn8AgiDown_22 AT %MX31232.22 : BOOL;
	bSlowPull2LifterStn8AgiDown_23 AT %MX31232.23 : BOOL;
	bSlowPull2LifterStn8AgiDown_24 AT %MX31232.24 : BOOL;
	bSlowPull2LifterStn8AgiDown_25 AT %MX31232.25 : BOOL;
	bSlowPull2LifterStn8AgiDown_26 AT %MX31232.26 : BOOL;
	bSlowPull2LifterStn8AgiDown_27 AT %MX31232.27 : BOOL;
	bSlowPull2LifterStn8AgiDown_28 AT %MX31232.28 : BOOL;
	bSlowPull2LifterStn8AgiDown_29 AT %MX31232.29 : BOOL;
	bSlowPull2LifterStn8AgiDown_30 AT %MX31232.30 : BOOL;
	bSlowPull2LifterStn8AgiDown_31 AT %MX31232.31 : BOOL;

	bSlowPull2LifterStn9AgiDown_00 AT %MX31236.0 : BOOL;
	bSlowPull2LifterStn9AgiDown_01 AT %MX31236.1 : BOOL;
	bSlowPull2LifterStn9AgiDown_02 AT %MX31236.2 : BOOL;
	bSlowPull2LifterStn9AgiDown_03 AT %MX31236.3 : BOOL;
	bSlowPull2LifterStn9AgiDown_04 AT %MX31236.4 : BOOL;
	bSlowPull2LifterStn9AgiDown_05 AT %MX31236.5 : BOOL;
	bSlowPull2LifterStn9AgiDown_06 AT %MX31236.6 : BOOL;
	bSlowPull2LifterStn9AgiDown_07 AT %MX31236.7 : BOOL;
	bSlowPull2LifterStn9AgiDown_08 AT %MX31236.8 : BOOL;
	bSlowPull2LifterStn9AgiDown_09 AT %MX31236.9 : BOOL;
	bSlowPull2LifterStn9AgiDown_10 AT %MX31236.10 : BOOL;
	bSlowPull2LifterStn9AgiDown_11 AT %MX31236.11 : BOOL;
	bSlowPull2LifterStn9AgiDown_12 AT %MX31236.12 : BOOL;
	bSlowPull2LifterStn9AgiDown_13 AT %MX31236.13 : BOOL;
	bSlowPull2LifterStn9AgiDown_14 AT %MX31236.14 : BOOL;
	bSlowPull2LifterStn9AgiDown_15 AT %MX31236.15 : BOOL;
	bSlowPull2LifterStn9AgiDown_16 AT %MX31236.16 : BOOL;
	bSlowPull2LifterStn9AgiDown_17 AT %MX31236.17 : BOOL;
	bSlowPull2LifterStn9AgiDown_18 AT %MX31236.18 : BOOL;
	bSlowPull2LifterStn9AgiDown_19 AT %MX31236.19 : BOOL;
	bSlowPull2LifterStn9AgiDown_20 AT %MX31236.20 : BOOL;
	bSlowPull2LifterStn9AgiDown_21 AT %MX31236.21 : BOOL;
	bSlowPull2LifterStn9AgiDown_22 AT %MX31236.22 : BOOL;
	bSlowPull2LifterStn9AgiDown_23 AT %MX31236.23 : BOOL;
	bSlowPull2LifterStn9AgiDown_24 AT %MX31236.24 : BOOL;
	bSlowPull2LifterStn9AgiDown_25 AT %MX31236.25 : BOOL;
	bSlowPull2LifterStn9AgiDown_26 AT %MX31236.26 : BOOL;
	bSlowPull2LifterStn9AgiDown_27 AT %MX31236.27 : BOOL;
	bSlowPull2LifterStn9AgiDown_28 AT %MX31236.28 : BOOL;
	bSlowPull2LifterStn9AgiDown_29 AT %MX31236.29 : BOOL;
	bSlowPull2LifterStn9AgiDown_30 AT %MX31236.30 : BOOL;
	bSlowPull2LifterStn9AgiDown_31 AT %MX31236.31 : BOOL;

	bSlowPull2LifterStn10AgiDown_00 AT %MX31240.0 : BOOL;
	bSlowPull2LifterStn10AgiDown_01 AT %MX31240.1 : BOOL;
	bSlowPull2LifterStn10AgiDown_02 AT %MX31240.2 : BOOL;
	bSlowPull2LifterStn10AgiDown_03 AT %MX31240.3 : BOOL;
	bSlowPull2LifterStn10AgiDown_04 AT %MX31240.4 : BOOL;
	bSlowPull2LifterStn10AgiDown_05 AT %MX31240.5 : BOOL;
	bSlowPull2LifterStn10AgiDown_06 AT %MX31240.6 : BOOL;
	bSlowPull2LifterStn10AgiDown_07 AT %MX31240.7 : BOOL;
	bSlowPull2LifterStn10AgiDown_08 AT %MX31240.8 : BOOL;
	bSlowPull2LifterStn10AgiDown_09 AT %MX31240.9 : BOOL;
	bSlowPull2LifterStn10AgiDown_10 AT %MX31240.10 : BOOL;
	bSlowPull2LifterStn10AgiDown_11 AT %MX31240.11 : BOOL;
	bSlowPull2LifterStn10AgiDown_12 AT %MX31240.12 : BOOL;
	bSlowPull2LifterStn10AgiDown_13 AT %MX31240.13 : BOOL;
	bSlowPull2LifterStn10AgiDown_14 AT %MX31240.14 : BOOL;
	bSlowPull2LifterStn10AgiDown_15 AT %MX31240.15 : BOOL;
	bSlowPull2LifterStn10AgiDown_16 AT %MX31240.16 : BOOL;
	bSlowPull2LifterStn10AgiDown_17 AT %MX31240.17 : BOOL;
	bSlowPull2LifterStn10AgiDown_18 AT %MX31240.18 : BOOL;
	bSlowPull2LifterStn10AgiDown_19 AT %MX31240.19 : BOOL;
	bSlowPull2LifterStn10AgiDown_20 AT %MX31240.20 : BOOL;
	bSlowPull2LifterStn10AgiDown_21 AT %MX31240.21 : BOOL;
	bSlowPull2LifterStn10AgiDown_22 AT %MX31240.22 : BOOL;
	bSlowPull2LifterStn10AgiDown_23 AT %MX31240.23 : BOOL;
	bSlowPull2LifterStn10AgiDown_24 AT %MX31240.24 : BOOL;
	bSlowPull2LifterStn10AgiDown_25 AT %MX31240.25 : BOOL;
	bSlowPull2LifterStn10AgiDown_26 AT %MX31240.26 : BOOL;
	bSlowPull2LifterStn10AgiDown_27 AT %MX31240.27 : BOOL;
	bSlowPull2LifterStn10AgiDown_28 AT %MX31240.28 : BOOL;
	bSlowPull2LifterStn10AgiDown_29 AT %MX31240.29 : BOOL;
	bSlowPull2LifterStn10AgiDown_30 AT %MX31240.30 : BOOL;
	bSlowPull2LifterStn10AgiDown_31 AT %MX31240.31 : BOOL;

	bSlowPull2LifterStn11AgiDown_00 AT %MX31244.0 : BOOL;
	bSlowPull2LifterStn11AgiDown_01 AT %MX31244.1 : BOOL;
	bSlowPull2LifterStn11AgiDown_02 AT %MX31244.2 : BOOL;
	bSlowPull2LifterStn11AgiDown_03 AT %MX31244.3 : BOOL;
	bSlowPull2LifterStn11AgiDown_04 AT %MX31244.4 : BOOL;
	bSlowPull2LifterStn11AgiDown_05 AT %MX31244.5 : BOOL;
	bSlowPull2LifterStn11AgiDown_06 AT %MX31244.6 : BOOL;
	bSlowPull2LifterStn11AgiDown_07 AT %MX31244.7 : BOOL;
	bSlowPull2LifterStn11AgiDown_08 AT %MX31244.8 : BOOL;
	bSlowPull2LifterStn11AgiDown_09 AT %MX31244.9 : BOOL;
	bSlowPull2LifterStn11AgiDown_10 AT %MX31244.10 : BOOL;
	bSlowPull2LifterStn11AgiDown_11 AT %MX31244.11 : BOOL;
	bSlowPull2LifterStn11AgiDown_12 AT %MX31244.12 : BOOL;
	bSlowPull2LifterStn11AgiDown_13 AT %MX31244.13 : BOOL;
	bSlowPull2LifterStn11AgiDown_14 AT %MX31244.14 : BOOL;
	bSlowPull2LifterStn11AgiDown_15 AT %MX31244.15 : BOOL;
	bSlowPull2LifterStn11AgiDown_16 AT %MX31244.16 : BOOL;
	bSlowPull2LifterStn11AgiDown_17 AT %MX31244.17 : BOOL;
	bSlowPull2LifterStn11AgiDown_18 AT %MX31244.18 : BOOL;
	bSlowPull2LifterStn11AgiDown_19 AT %MX31244.19 : BOOL;
	bSlowPull2LifterStn11AgiDown_20 AT %MX31244.20 : BOOL;
	bSlowPull2LifterStn11AgiDown_21 AT %MX31244.21 : BOOL;
	bSlowPull2LifterStn11AgiDown_22 AT %MX31244.22 : BOOL;
	bSlowPull2LifterStn11AgiDown_23 AT %MX31244.23 : BOOL;
	bSlowPull2LifterStn11AgiDown_24 AT %MX31244.24 : BOOL;
	bSlowPull2LifterStn11AgiDown_25 AT %MX31244.25 : BOOL;
	bSlowPull2LifterStn11AgiDown_26 AT %MX31244.26 : BOOL;
	bSlowPull2LifterStn11AgiDown_27 AT %MX31244.27 : BOOL;
	bSlowPull2LifterStn11AgiDown_28 AT %MX31244.28 : BOOL;
	bSlowPull2LifterStn11AgiDown_29 AT %MX31244.29 : BOOL;
	bSlowPull2LifterStn11AgiDown_30 AT %MX31244.30 : BOOL;
	bSlowPull2LifterStn11AgiDown_31 AT %MX31244.31 : BOOL;

	bSlowPull2LifterStn12AgiDown_00 AT %MX31248.0 : BOOL;
	bSlowPull2LifterStn12AgiDown_01 AT %MX31248.1 : BOOL;
	bSlowPull2LifterStn12AgiDown_02 AT %MX31248.2 : BOOL;
	bSlowPull2LifterStn12AgiDown_03 AT %MX31248.3 : BOOL;
	bSlowPull2LifterStn12AgiDown_04 AT %MX31248.4 : BOOL;
	bSlowPull2LifterStn12AgiDown_05 AT %MX31248.5 : BOOL;
	bSlowPull2LifterStn12AgiDown_06 AT %MX31248.6 : BOOL;
	bSlowPull2LifterStn12AgiDown_07 AT %MX31248.7 : BOOL;
	bSlowPull2LifterStn12AgiDown_08 AT %MX31248.8 : BOOL;
	bSlowPull2LifterStn12AgiDown_09 AT %MX31248.9 : BOOL;
	bSlowPull2LifterStn12AgiDown_10 AT %MX31248.10 : BOOL;
	bSlowPull2LifterStn12AgiDown_11 AT %MX31248.11 : BOOL;
	bSlowPull2LifterStn12AgiDown_12 AT %MX31248.12 : BOOL;
	bSlowPull2LifterStn12AgiDown_13 AT %MX31248.13 : BOOL;
	bSlowPull2LifterStn12AgiDown_14 AT %MX31248.14 : BOOL;
	bSlowPull2LifterStn12AgiDown_15 AT %MX31248.15 : BOOL;
	bSlowPull2LifterStn12AgiDown_16 AT %MX31248.16 : BOOL;
	bSlowPull2LifterStn12AgiDown_17 AT %MX31248.17 : BOOL;
	bSlowPull2LifterStn12AgiDown_18 AT %MX31248.18 : BOOL;
	bSlowPull2LifterStn12AgiDown_19 AT %MX31248.19 : BOOL;
	bSlowPull2LifterStn12AgiDown_20 AT %MX31248.20 : BOOL;
	bSlowPull2LifterStn12AgiDown_21 AT %MX31248.21 : BOOL;
	bSlowPull2LifterStn12AgiDown_22 AT %MX31248.22 : BOOL;
	bSlowPull2LifterStn12AgiDown_23 AT %MX31248.23 : BOOL;
	bSlowPull2LifterStn12AgiDown_24 AT %MX31248.24 : BOOL;
	bSlowPull2LifterStn12AgiDown_25 AT %MX31248.25 : BOOL;
	bSlowPull2LifterStn12AgiDown_26 AT %MX31248.26 : BOOL;
	bSlowPull2LifterStn12AgiDown_27 AT %MX31248.27 : BOOL;
	bSlowPull2LifterStn12AgiDown_28 AT %MX31248.28 : BOOL;
	bSlowPull2LifterStn12AgiDown_29 AT %MX31248.29 : BOOL;
	bSlowPull2LifterStn12AgiDown_30 AT %MX31248.30 : BOOL;
	bSlowPull2LifterStn12AgiDown_31 AT %MX31248.31 : BOOL;


END_VAR

(* stored: Version 1.1.0.1, ProductVersion 3.1.4024.12
   GVL Global_Variables_Arm2BoolCtrl: Id {f6e93c0b-b904-4ae9-8643-4e26659c5b8d} *)
